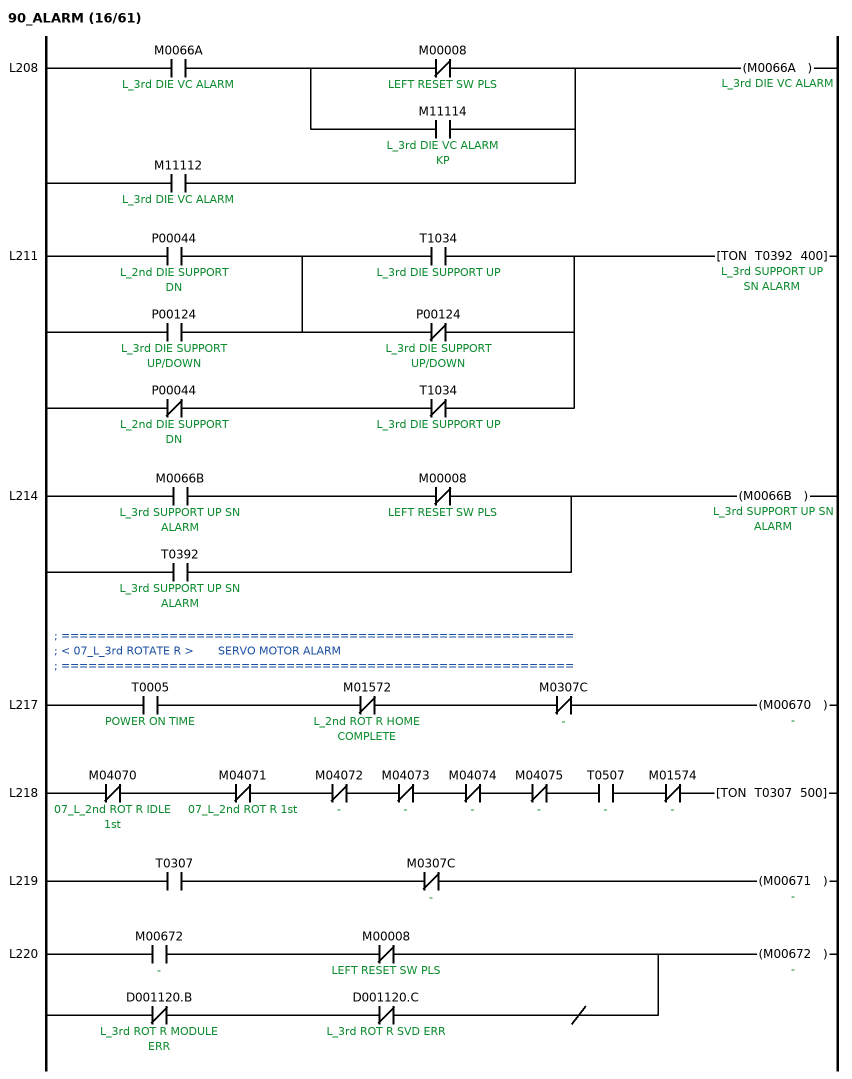
[picture p384: 90_ALARM rungs L208-L220]
; L208
LOAD      M0066A	// L_3rd DIE VC ALARM
LOAD NOT  M00008	// LEFT RESET SW PLS
OR        M11114	// L_3rd DIE VC ALARM KP
AND LOAD
OR        M11112	// L_3rd DIE VC ALARM
OUT       M0066A	// L_3rd DIE VC ALARM
; L211
LOAD      P00044	// L_2nd DIE SUPPORT DN
OR        P00124	// L_3rd DIE SUPPORT UP/DOWN
LOAD      T1034	// L_3rd DIE SUPPORT UP
OR NOT    P00124	// L_3rd DIE SUPPORT UP/DOWN
AND LOAD
LOAD NOT  P00044	// L_2nd DIE SUPPORT DN
AND NOT   T1034	// L_3rd DIE SUPPORT UP
OR LOAD
TON       T0392 400	// L_3rd SUPPORT UP SN ALARM
; L214
LOAD      M0066B	// L_3rd SUPPORT UP SN ALARM
AND NOT   M00008	// LEFT RESET SW PLS
OR        T0392	// L_3rd SUPPORT UP SN ALARM
OUT       M0066B	// L_3rd SUPPORT UP SN ALARM
// =========================================================
// 
//        < 07_L_3rd ROTATE R >       SERVO MOTOR ALARM
// 
// =========================================================
; L217
LOAD      T0005	// POWER ON TIME
AND NOT   M01572	// L_2nd ROT R HOME COMPLETE
AND NOT   M0307C	// -
OUT       M00670	// -
; L218
LOAD NOT  M04070	// 07_L_2nd ROT R IDLE 1st
AND NOT   M04071	// 07_L_2nd ROT R 1st
AND NOT   M04072	// -
AND NOT   M04073	// -
AND NOT   M04074	// -
AND NOT   M04075	// -
AND       T0507	// -
AND NOT   M01574	// -
TON       T0307 500
; L219
LOAD      T0307
AND NOT   M0307C	// -
OUT       M00671	// -
; L220
LOAD      M00672	// -
AND NOT   M00008	// LEFT RESET SW PLS
LOAD NOT  D001120.B	// L_3rd ROT R MODULE ERR
AND NOT   D001120.C	// L_3rd ROT R SVD ERR
NOT
OR LOAD
OUT       M00672	// -

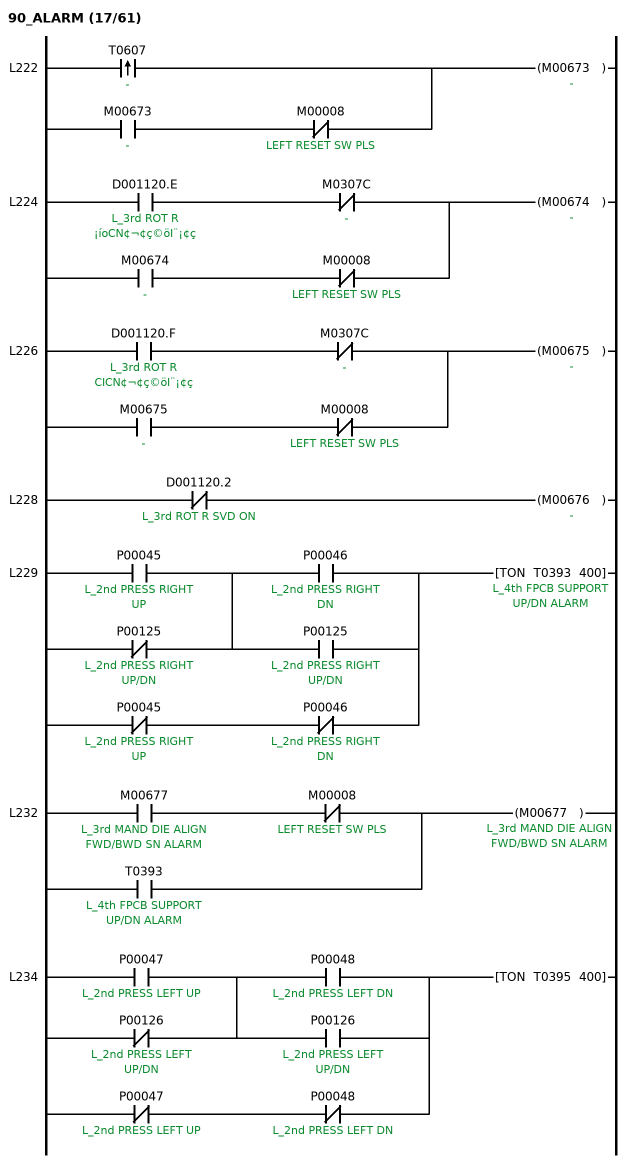
; L222
LOADP     T0607	// -
LOAD      M00673	// -
AND NOT   M00008	// LEFT RESET SW PLS
OR LOAD
OUT       M00673	// -
; L224
LOAD      D001120.E	// L_3rd ROT R ¡íoCN¢¬¢ç©öI¨¡¢ç
AND NOT   M0307C	// -
LOAD      M00674	// -
AND NOT   M00008	// LEFT RESET SW PLS
OR LOAD
OUT       M00674	// -
; L226
LOAD      D001120.F	// L_3rd ROT R CICN¢¬¢ç©öI¨¡¢ç
AND NOT   M0307C	// -
LOAD      M00675	// -
AND NOT   M00008	// LEFT RESET SW PLS
OR LOAD
OUT       M00675	// -
; L228
LOAD NOT  D001120.2	// L_3rd ROT R SVD ON
OUT       M00676	// -
; L229
LOAD      P00045	// L_2nd PRESS RIGHT UP
OR NOT    P00125	// L_2nd PRESS RIGHT UP/DN
LOAD      P00046	// L_2nd PRESS RIGHT DN
OR        P00125	// L_2nd PRESS RIGHT UP/DN
AND LOAD
LOAD NOT  P00045	// L_2nd PRESS RIGHT UP
AND NOT   P00046	// L_2nd PRESS RIGHT DN
OR LOAD
TON       T0393 400	// L_4th FPCB SUPPORT UP/DN ALARM
; L232
LOAD      M00677	// L_3rd MAND DIE ALIGN FWD/BWD SN ALARM
AND NOT   M00008	// LEFT RESET SW PLS
OR        T0393	// L_4th FPCB SUPPORT UP/DN ALARM
OUT       M00677	// L_3rd MAND DIE ALIGN FWD/BWD SN ALARM
; L234
LOAD      P00047	// L_2nd PRESS LEFT UP
OR NOT    P00126	// L_2nd PRESS LEFT UP/DN
LOAD      P00048	// L_2nd PRESS LEFT DN
OR        P00126	// L_2nd PRESS LEFT UP/DN
AND LOAD
LOAD NOT  P00047	// L_2nd PRESS LEFT UP
AND NOT   P00048	// L_2nd PRESS LEFT DN
OR LOAD
TON       T0395 400

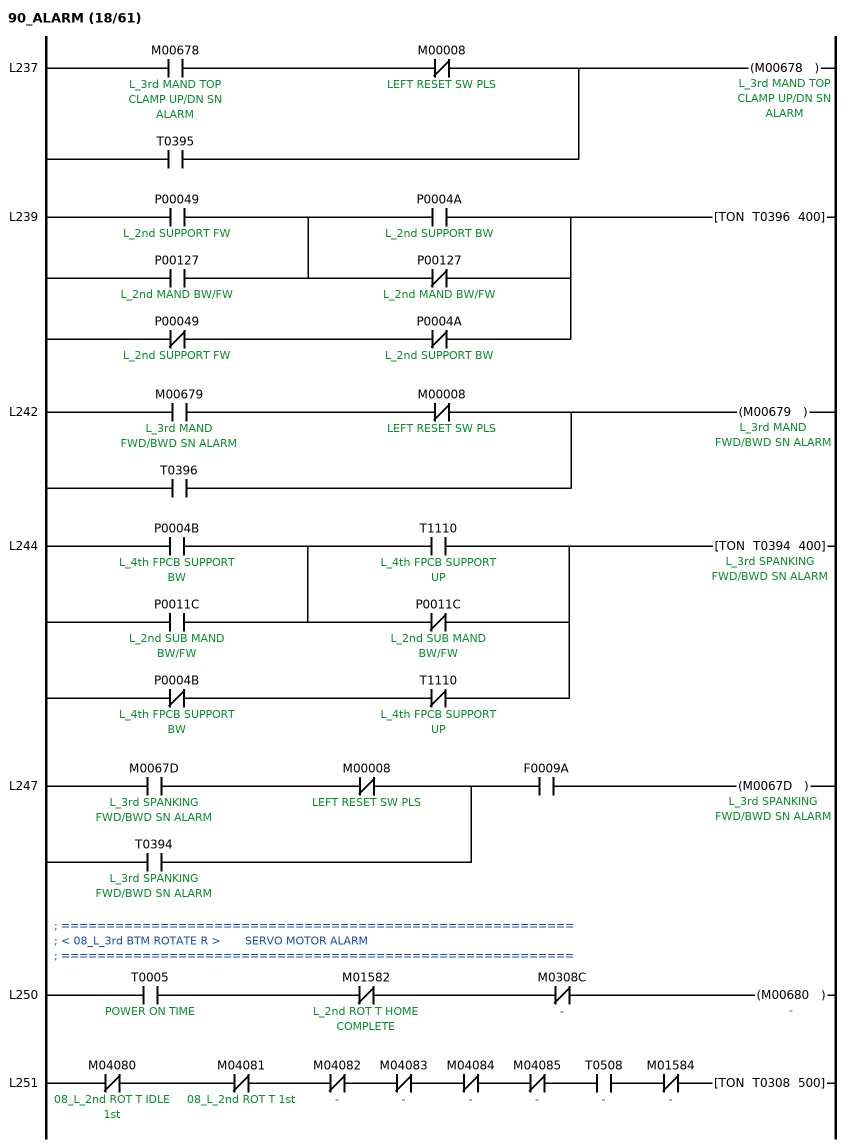
; L237
LOAD      M00678	// L_3rd MAND TOP CLAMP UP/DN SN ALARM
AND NOT   M00008	// LEFT RESET SW PLS
OR        T0395
OUT       M00678	// L_3rd MAND TOP CLAMP UP/DN SN ALARM
; L239
LOAD      P00049	// L_2nd SUPPORT FW
OR        P00127	// L_2nd MAND BW/FW
LOAD      P0004A	// L_2nd SUPPORT BW
OR NOT    P00127	// L_2nd MAND BW/FW
AND LOAD
LOAD NOT  P00049	// L_2nd SUPPORT FW
AND NOT   P0004A	// L_2nd SUPPORT BW
OR LOAD
TON       T0396 400
; L242
LOAD      M00679	// L_3rd MAND FWD/BWD SN ALARM
AND NOT   M00008	// LEFT RESET SW PLS
OR        T0396
OUT       M00679	// L_3rd MAND FWD/BWD SN ALARM
; L244
LOAD      P0004B	// L_4th FPCB SUPPORT BW
OR        P0011C	// L_2nd SUB MAND BW/FW
LOAD      T1110	// L_4th FPCB SUPPORT UP
OR NOT    P0011C	// L_2nd SUB MAND BW/FW
AND LOAD
LOAD NOT  P0004B	// L_4th FPCB SUPPORT BW
AND NOT   T1110	// L_4th FPCB SUPPORT UP
OR LOAD
TON       T0394 400	// L_3rd SPANKING FWD/BWD SN ALARM
; L247
LOAD      M0067D	// L_3rd SPANKING FWD/BWD SN ALARM
AND NOT   M00008	// LEFT RESET SW PLS
OR        T0394	// L_3rd SPANKING FWD/BWD SN ALARM
AND       F0009A
OUT       M0067D	// L_3rd SPANKING FWD/BWD SN ALARM
// =========================================================
// 
//        < 08_L_3rd BTM ROTATE R >       SERVO MOTOR ALARM
// 
// =========================================================
; L250
LOAD      T0005	// POWER ON TIME
AND NOT   M01582	// L_2nd ROT T HOME COMPLETE
AND NOT   M0308C	// -
OUT       M00680	// -
; L251
LOAD NOT  M04080	// 08_L_2nd ROT T IDLE 1st
AND NOT   M04081	// 08_L_2nd ROT T 1st
AND NOT   M04082	// -
AND NOT   M04083	// -
AND NOT   M04084	// -
AND NOT   M04085	// -
AND       T0508	// -
AND NOT   M01584	// -
TON       T0308 500

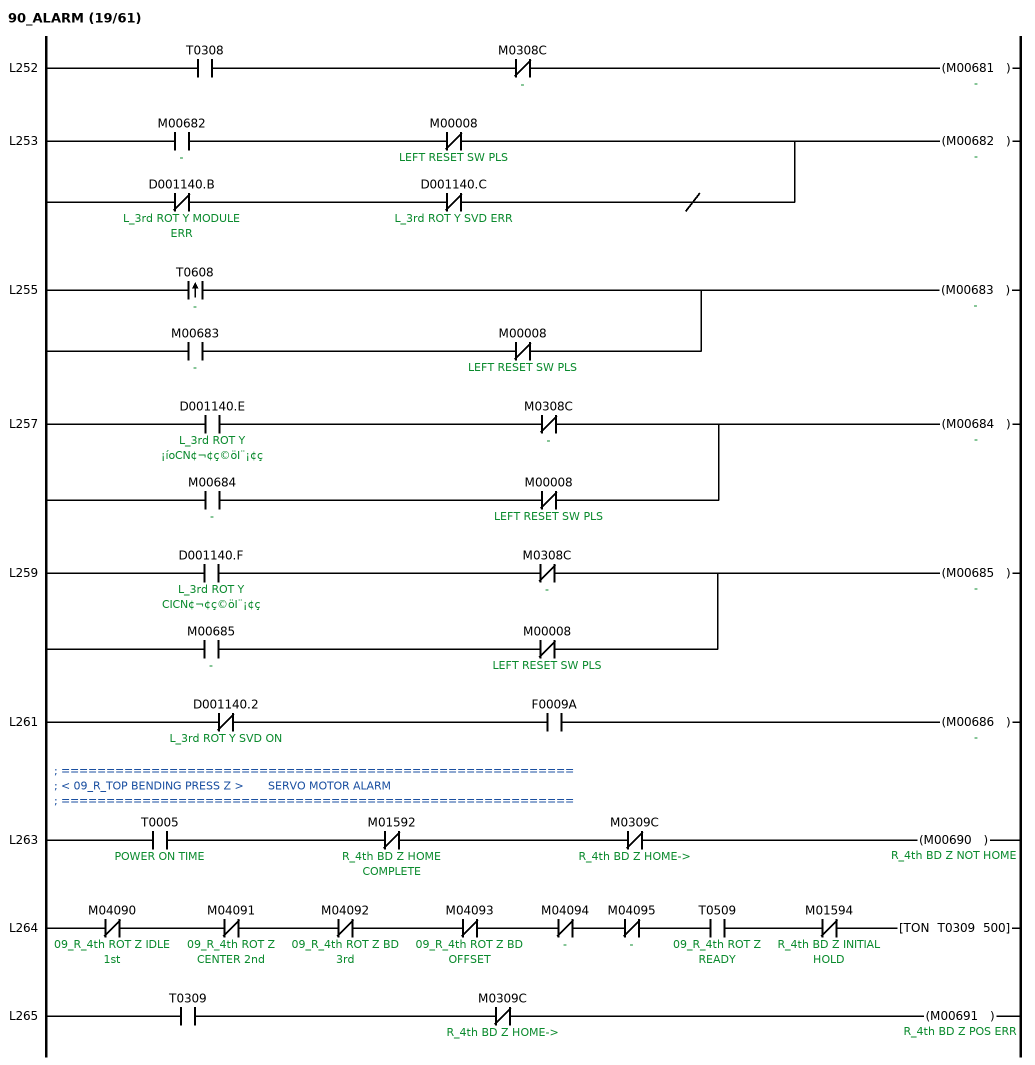
; L252
LOAD      T0308
AND NOT   M0308C	// -
OUT       M00681	// -
; L253
LOAD      M00682	// -
AND NOT   M00008	// LEFT RESET SW PLS
LOAD NOT  D001140.B	// L_3rd ROT Y MODULE ERR
AND NOT   D001140.C	// L_3rd ROT Y SVD ERR
NOT
OR LOAD
OUT       M00682	// -
; L255
LOADP     T0608	// -
LOAD      M00683	// -
AND NOT   M00008	// LEFT RESET SW PLS
OR LOAD
OUT       M00683	// -
; L257
LOAD      D001140.E	// L_3rd ROT Y ¡íoCN¢¬¢ç©öI¨¡¢ç
AND NOT   M0308C	// -
LOAD      M00684	// -
AND NOT   M00008	// LEFT RESET SW PLS
OR LOAD
OUT       M00684	// -
; L259
LOAD      D001140.F	// L_3rd ROT Y CICN¢¬¢ç©öI¨¡¢ç
AND NOT   M0308C	// -
LOAD      M00685	// -
AND NOT   M00008	// LEFT RESET SW PLS
OR LOAD
OUT       M00685	// -
; L261
LOAD NOT  D001140.2	// L_3rd ROT Y SVD ON
AND       F0009A
OUT       M00686	// -
// =========================================================
// 
//        < 09_R_TOP BENDING PRESS Z >       SERVO MOTOR ALARM
// 
// =========================================================
; L263
LOAD      T0005	// POWER ON TIME
AND NOT   M01592	// R_4th BD Z HOME COMPLETE
AND NOT   M0309C	// R_4th BD Z HOME->
OUT       M00690	// R_4th BD Z NOT HOME
; L264
LOAD NOT  M04090	// 09_R_4th ROT Z IDLE 1st
AND NOT   M04091	// 09_R_4th ROT Z CENTER 2nd
AND NOT   M04092	// 09_R_4th ROT Z BD 3rd
AND NOT   M04093	// 09_R_4th ROT Z BD OFFSET
AND NOT   M04094	// -
AND NOT   M04095	// -
AND       T0509	// 09_R_4th ROT Z READY
AND NOT   M01594	// R_4th BD Z INITIAL HOLD
TON       T0309 500
; L265
LOAD      T0309
AND NOT   M0309C	// R_4th BD Z HOME->
OUT       M00691	// R_4th BD Z POS ERR

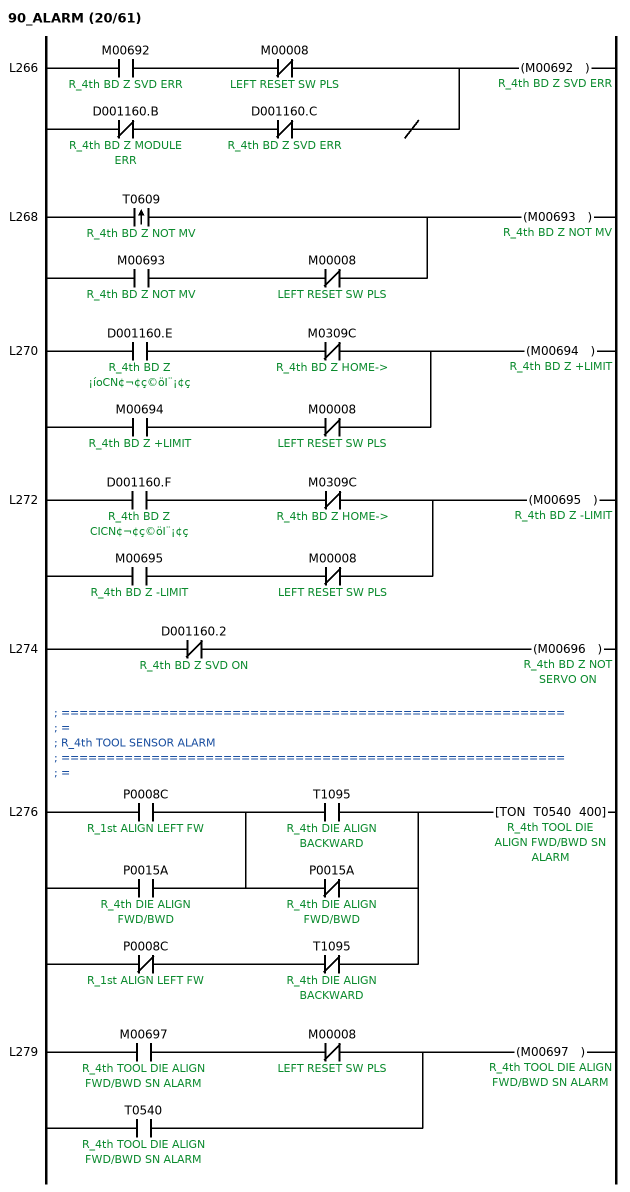
; L266
LOAD      M00692	// R_4th BD Z SVD ERR
AND NOT   M00008	// LEFT RESET SW PLS
LOAD NOT  D001160.B	// R_4th BD Z MODULE ERR
AND NOT   D001160.C	// R_4th BD Z SVD ERR
NOT
OR LOAD
OUT       M00692	// R_4th BD Z SVD ERR
; L268
LOADP     T0609	// R_4th BD Z NOT MV
LOAD      M00693	// R_4th BD Z NOT MV
AND NOT   M00008	// LEFT RESET SW PLS
OR LOAD
OUT       M00693	// R_4th BD Z NOT MV
; L270
LOAD      D001160.E	// R_4th BD Z ¡íoCN¢¬¢ç©öI¨¡¢ç
AND NOT   M0309C	// R_4th BD Z HOME->
LOAD      M00694	// R_4th BD Z +LIMIT
AND NOT   M00008	// LEFT RESET SW PLS
OR LOAD
OUT       M00694	// R_4th BD Z +LIMIT
; L272
LOAD      D001160.F	// R_4th BD Z CICN¢¬¢ç©öI¨¡¢ç
AND NOT   M0309C	// R_4th BD Z HOME->
LOAD      M00695	// R_4th BD Z -LIMIT
AND NOT   M00008	// LEFT RESET SW PLS
OR LOAD
OUT       M00695	// R_4th BD Z -LIMIT
; L274
LOAD NOT  D001160.2	// R_4th BD Z SVD ON
OUT       M00696	// R_4th BD Z NOT SERVO ON
// =========================================================
// 
//        R_4th TOOL SENSOR ALARM
// 
// =========================================================
; L276
LOAD      P0008C	// R_1st ALIGN LEFT FW
OR        P0015A	// R_4th DIE ALIGN FWD/BWD
LOAD      T1095	// R_4th DIE ALIGN BACKWARD
OR NOT    P0015A	// R_4th DIE ALIGN FWD/BWD
AND LOAD
LOAD NOT  P0008C	// R_1st ALIGN LEFT FW
AND NOT   T1095	// R_4th DIE ALIGN BACKWARD
OR LOAD
TON       T0540 400	// R_4th TOOL DIE ALIGN FWD/BWD SN ALARM
; L279
LOAD      M00697	// R_4th TOOL DIE ALIGN FWD/BWD SN ALARM
AND NOT   M00008	// LEFT RESET SW PLS
OR        T0540	// R_4th TOOL DIE ALIGN FWD/BWD SN ALARM
OUT       M00697	// R_4th TOOL DIE ALIGN FWD/BWD SN ALARM

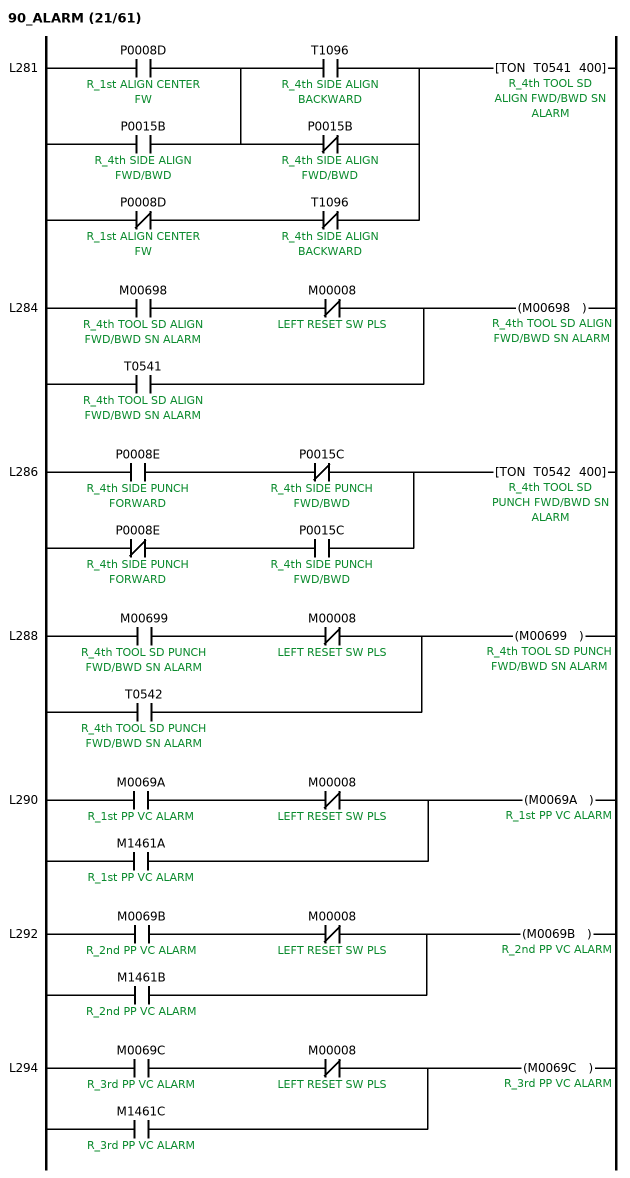
; L281
LOAD      P0008D	// R_1st ALIGN CENTER FW
OR        P0015B	// R_4th SIDE ALIGN FWD/BWD
LOAD      T1096	// R_4th SIDE ALIGN BACKWARD
OR NOT    P0015B	// R_4th SIDE ALIGN FWD/BWD
AND LOAD
LOAD NOT  P0008D	// R_1st ALIGN CENTER FW
AND NOT   T1096	// R_4th SIDE ALIGN BACKWARD
OR LOAD
TON       T0541 400	// R_4th TOOL SD ALIGN FWD/BWD SN ALARM
; L284
LOAD      M00698	// R_4th TOOL SD ALIGN FWD/BWD SN ALARM
AND NOT   M00008	// LEFT RESET SW PLS
OR        T0541	// R_4th TOOL SD ALIGN FWD/BWD SN ALARM
OUT       M00698	// R_4th TOOL SD ALIGN FWD/BWD SN ALARM
; L286
LOAD      P0008E	// R_4th SIDE PUNCH FORWARD
AND NOT   P0015C	// R_4th SIDE PUNCH FWD/BWD
LOAD NOT  P0008E	// R_4th SIDE PUNCH FORWARD
AND       P0015C	// R_4th SIDE PUNCH FWD/BWD
OR LOAD
TON       T0542 400	// R_4th TOOL SD PUNCH FWD/BWD SN ALARM
; L288
LOAD      M00699	// R_4th TOOL SD PUNCH FWD/BWD SN ALARM
AND NOT   M00008	// LEFT RESET SW PLS
OR        T0542	// R_4th TOOL SD PUNCH FWD/BWD SN ALARM
OUT       M00699	// R_4th TOOL SD PUNCH FWD/BWD SN ALARM
; L290
LOAD      M0069A	// R_1st PP VC ALARM
AND NOT   M00008	// LEFT RESET SW PLS
OR        M1461A	// R_1st PP VC ALARM
OUT       M0069A	// R_1st PP VC ALARM
; L292
LOAD      M0069B	// R_2nd PP VC ALARM
AND NOT   M00008	// LEFT RESET SW PLS
OR        M1461B	// R_2nd PP VC ALARM
OUT       M0069B	// R_2nd PP VC ALARM
; L294
LOAD      M0069C	// R_3rd PP VC ALARM
AND NOT   M00008	// LEFT RESET SW PLS
OR        M1461C	// R_3rd PP VC ALARM
OUT       M0069C	// R_3rd PP VC ALARM

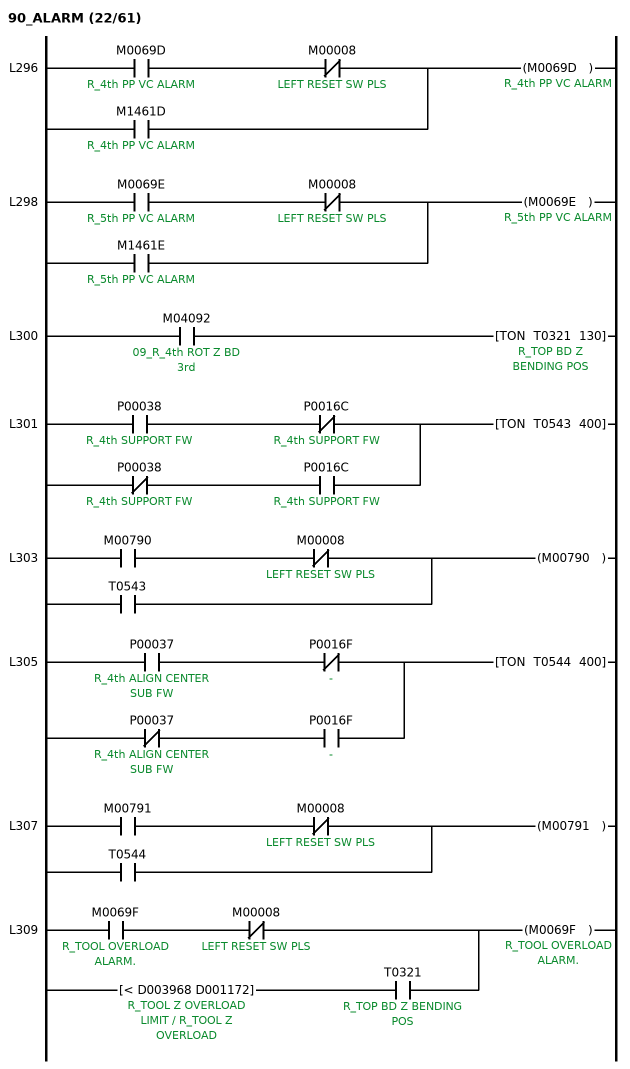
; L296
LOAD      M0069D	// R_4th PP VC ALARM
AND NOT   M00008	// LEFT RESET SW PLS
OR        M1461D	// R_4th PP VC ALARM
OUT       M0069D	// R_4th PP VC ALARM
; L298
LOAD      M0069E	// R_5th PP VC ALARM
AND NOT   M00008	// LEFT RESET SW PLS
OR        M1461E	// R_5th PP VC ALARM
OUT       M0069E	// R_5th PP VC ALARM
; L300
LOAD      M04092	// 09_R_4th ROT Z BD 3rd
TON       T0321 130	// R_TOP BD Z BENDING POS
; L301
LOAD      P00038	// R_4th SUPPORT FW
AND NOT   P0016C	// R_4th SUPPORT FW
LOAD NOT  P00038	// R_4th SUPPORT FW
AND       P0016C	// R_4th SUPPORT FW
OR LOAD
TON       T0543 400
; L303
LOAD      M00790
AND NOT   M00008	// LEFT RESET SW PLS
OR        T0543
OUT       M00790
; L305
LOAD      P00037	// R_4th ALIGN CENTER SUB FW
AND NOT   P0016F	// -
LOAD NOT  P00037	// R_4th ALIGN CENTER SUB FW
AND       P0016F	// -
OR LOAD
TON       T0544 400
; L307
LOAD      M00791
AND NOT   M00008	// LEFT RESET SW PLS
OR        T0544
OUT       M00791
; L309
LOAD      M0069F	// R_TOOL OVERLOAD ALARM.
AND NOT   M00008	// LEFT RESET SW PLS
LOAD<     D003968 D001172	// R_TOOL Z OVERLOAD LIMIT / R_TOOL Z OVERLOAD
AND       T0321	// R_TOP BD Z BENDING POS
OR LOAD
OUT       M0069F	// R_TOOL OVERLOAD ALARM.

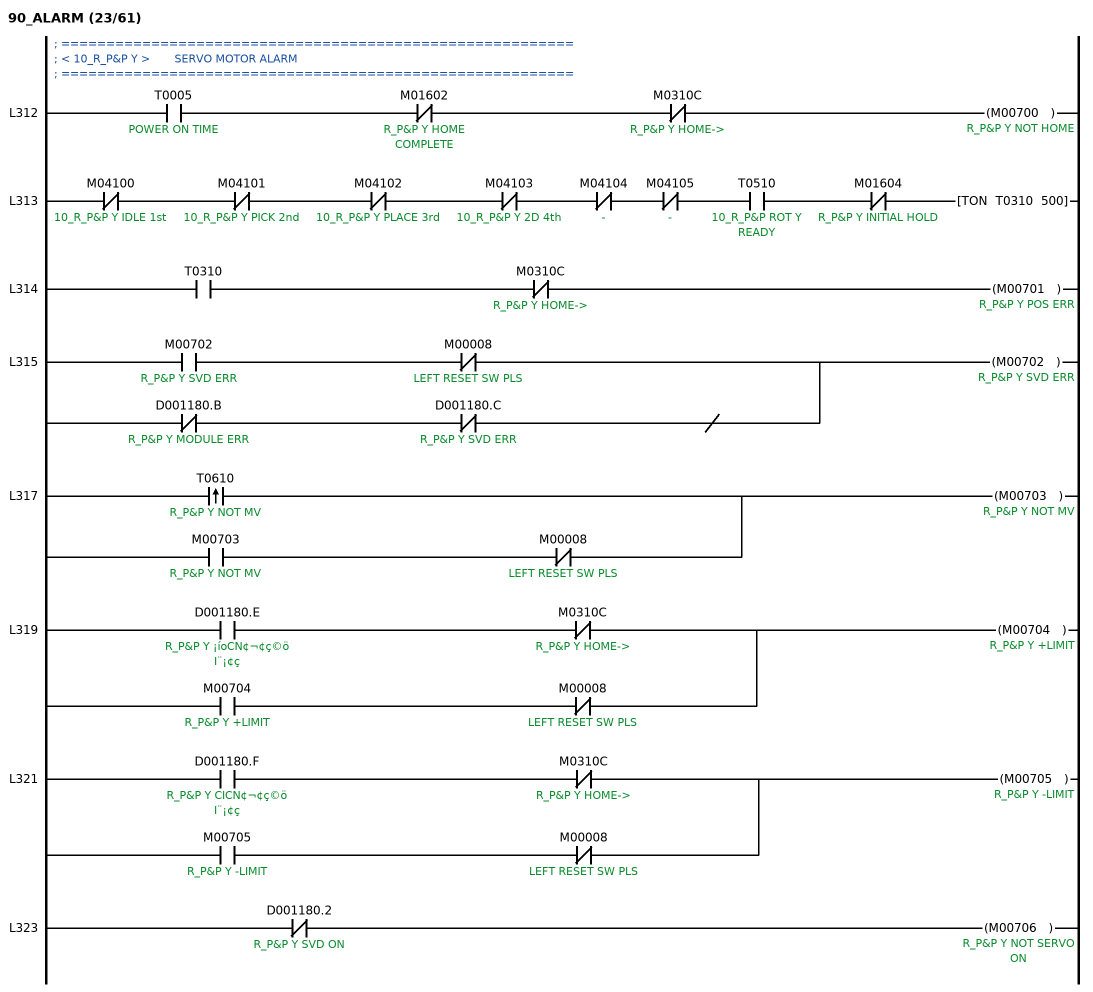
// =========================================================
// 
//        < 10_R_P&P Y >       SERVO MOTOR ALARM
// 
// =========================================================
; L312
LOAD      T0005	// POWER ON TIME
AND NOT   M01602	// R_P&P Y HOME COMPLETE
AND NOT   M0310C	// R_P&P Y HOME->
OUT       M00700	// R_P&P Y NOT HOME
; L313
LOAD NOT  M04100	// 10_R_P&P Y IDLE 1st
AND NOT   M04101	// 10_R_P&P Y PICK 2nd
AND NOT   M04102	// 10_R_P&P Y PLACE 3rd
AND NOT   M04103	// 10_R_P&P Y 2D 4th
AND NOT   M04104	// -
AND NOT   M04105	// -
AND       T0510	// 10_R_P&P ROT Y READY
AND NOT   M01604	// R_P&P Y INITIAL HOLD
TON       T0310 500
; L314
LOAD      T0310
AND NOT   M0310C	// R_P&P Y HOME->
OUT       M00701	// R_P&P Y POS ERR
; L315
LOAD      M00702	// R_P&P Y SVD ERR
AND NOT   M00008	// LEFT RESET SW PLS
LOAD NOT  D001180.B	// R_P&P Y MODULE ERR
AND NOT   D001180.C	// R_P&P Y SVD ERR
NOT
OR LOAD
OUT       M00702	// R_P&P Y SVD ERR
; L317
LOADP     T0610	// R_P&P Y NOT MV
LOAD      M00703	// R_P&P Y NOT MV
AND NOT   M00008	// LEFT RESET SW PLS
OR LOAD
OUT       M00703	// R_P&P Y NOT MV
; L319
LOAD      D001180.E	// R_P&P Y ¡íoCN¢¬¢ç©öI¨¡¢ç
AND NOT   M0310C	// R_P&P Y HOME->
LOAD      M00704	// R_P&P Y +LIMIT
AND NOT   M00008	// LEFT RESET SW PLS
OR LOAD
OUT       M00704	// R_P&P Y +LIMIT
; L321
LOAD      D001180.F	// R_P&P Y CICN¢¬¢ç©öI¨¡¢ç
AND NOT   M0310C	// R_P&P Y HOME->
LOAD      M00705	// R_P&P Y -LIMIT
AND NOT   M00008	// LEFT RESET SW PLS
OR LOAD
OUT       M00705	// R_P&P Y -LIMIT
; L323
LOAD NOT  D001180.2	// R_P&P Y SVD ON
OUT       M00706	// R_P&P Y NOT SERVO ON

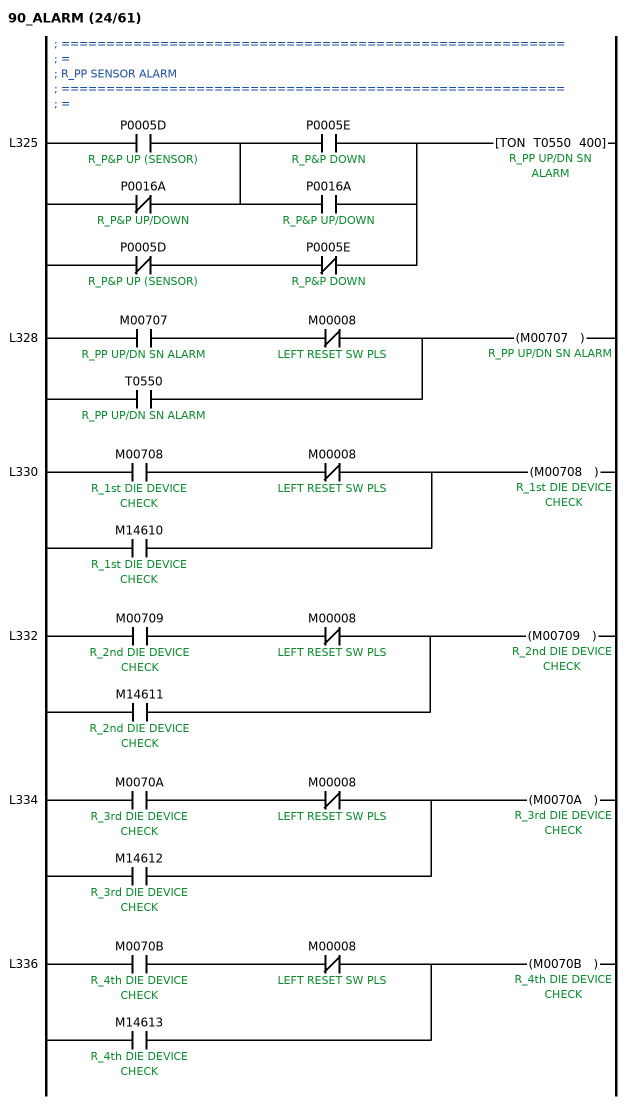
// =========================================================
// 
//       R_PP SENSOR ALARM
// 
// =========================================================
; L325
LOAD      P0005D	// R_P&P UP (SENSOR)
OR NOT    P0016A	// R_P&P UP/DOWN
LOAD      P0005E	// R_P&P DOWN
OR        P0016A	// R_P&P UP/DOWN
AND LOAD
LOAD NOT  P0005D	// R_P&P UP (SENSOR)
AND NOT   P0005E	// R_P&P DOWN
OR LOAD
TON       T0550 400	// R_PP UP/DN SN ALARM
; L328
LOAD      M00707	// R_PP UP/DN SN ALARM
AND NOT   M00008	// LEFT RESET SW PLS
OR        T0550	// R_PP UP/DN SN ALARM
OUT       M00707	// R_PP UP/DN SN ALARM
; L330
LOAD      M00708	// R_1st DIE DEVICE CHECK
AND NOT   M00008	// LEFT RESET SW PLS
OR        M14610	// R_1st DIE DEVICE CHECK
OUT       M00708	// R_1st DIE DEVICE CHECK
; L332
LOAD      M00709	// R_2nd DIE DEVICE CHECK
AND NOT   M00008	// LEFT RESET SW PLS
OR        M14611	// R_2nd DIE DEVICE CHECK
OUT       M00709	// R_2nd DIE DEVICE CHECK
; L334
LOAD      M0070A	// R_3rd DIE DEVICE CHECK
AND NOT   M00008	// LEFT RESET SW PLS
OR        M14612	// R_3rd DIE DEVICE CHECK
OUT       M0070A	// R_3rd DIE DEVICE CHECK
; L336
LOAD      M0070B	// R_4th DIE DEVICE CHECK
AND NOT   M00008	// LEFT RESET SW PLS
OR        M14613	// R_4th DIE DEVICE CHECK
OUT       M0070B	// R_4th DIE DEVICE CHECK

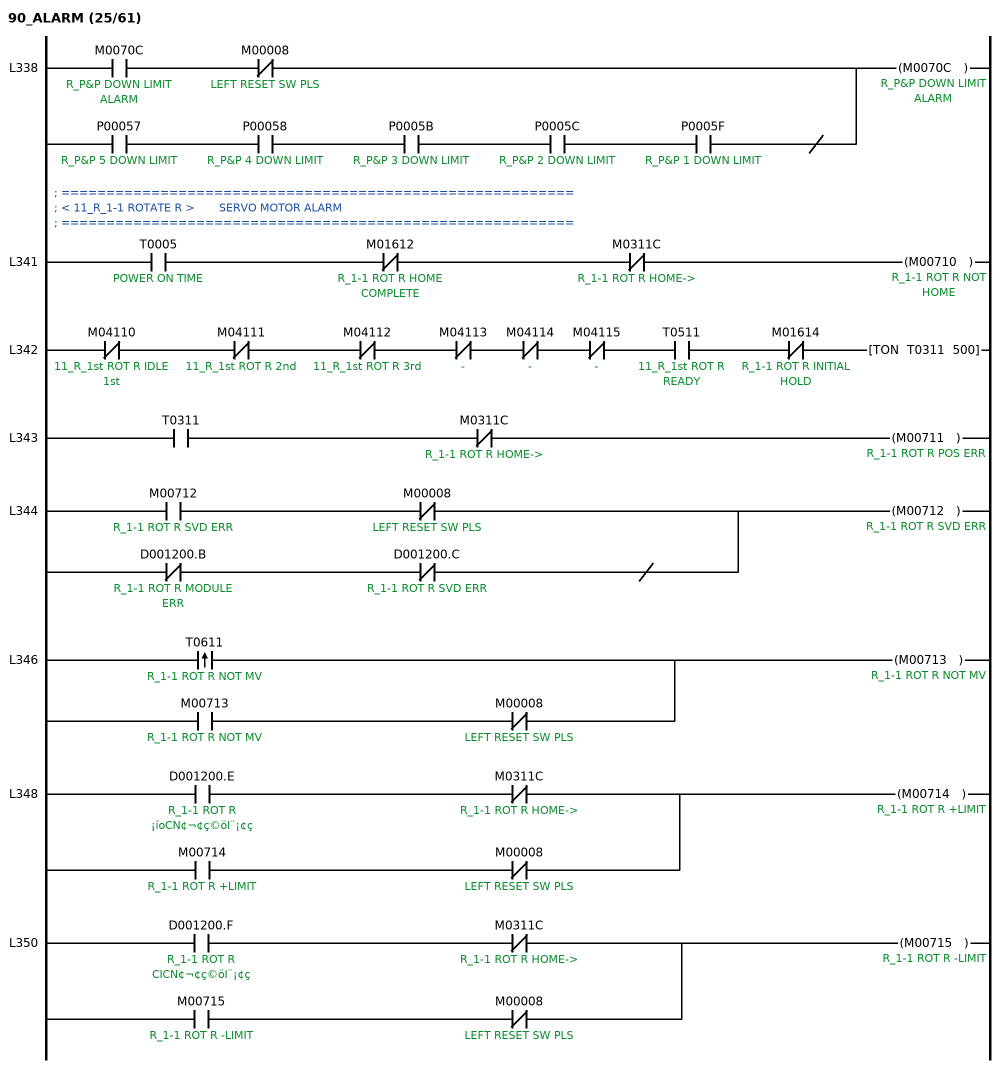
; L338
LOAD      M0070C	// R_P&P DOWN LIMIT ALARM
AND NOT   M00008	// LEFT RESET SW PLS
LOAD      P00057	// R_P&P 5 DOWN LIMIT
AND       P00058	// R_P&P 4 DOWN LIMIT
AND       P0005B	// R_P&P 3 DOWN LIMIT
AND       P0005C	// R_P&P 2 DOWN LIMIT
AND       P0005F	// R_P&P 1 DOWN LIMIT
NOT
OR LOAD
OUT       M0070C	// R_P&P DOWN LIMIT ALARM
// =========================================================
// 
//        < 11_R_1-1 ROTATE R >       SERVO MOTOR ALARM
// 
// =========================================================
; L341
LOAD      T0005	// POWER ON TIME
AND NOT   M01612	// R_1-1 ROT R HOME COMPLETE
AND NOT   M0311C	// R_1-1 ROT R HOME->
OUT       M00710	// R_1-1 ROT R NOT HOME
; L342
LOAD NOT  M04110	// 11_R_1st ROT R IDLE 1st
AND NOT   M04111	// 11_R_1st ROT R 2nd
AND NOT   M04112	// 11_R_1st ROT R 3rd
AND NOT   M04113	// -
AND NOT   M04114	// -
AND NOT   M04115	// -
AND       T0511	// 11_R_1st ROT R READY
AND NOT   M01614	// R_1-1 ROT R INITIAL HOLD
TON       T0311 500
; L343
LOAD      T0311
AND NOT   M0311C	// R_1-1 ROT R HOME->
OUT       M00711	// R_1-1 ROT R POS ERR
; L344
LOAD      M00712	// R_1-1 ROT R SVD ERR
AND NOT   M00008	// LEFT RESET SW PLS
LOAD NOT  D001200.B	// R_1-1 ROT R MODULE ERR
AND NOT   D001200.C	// R_1-1 ROT R SVD ERR
NOT
OR LOAD
OUT       M00712	// R_1-1 ROT R SVD ERR
; L346
LOADP     T0611	// R_1-1 ROT R NOT MV
LOAD      M00713	// R_1-1 ROT R NOT MV
AND NOT   M00008	// LEFT RESET SW PLS
OR LOAD
OUT       M00713	// R_1-1 ROT R NOT MV
; L348
LOAD      D001200.E	// R_1-1 ROT R ¡íoCN¢¬¢ç©öI¨¡¢ç
AND NOT   M0311C	// R_1-1 ROT R HOME->
LOAD      M00714	// R_1-1 ROT R +LIMIT
AND NOT   M00008	// LEFT RESET SW PLS
OR LOAD
OUT       M00714	// R_1-1 ROT R +LIMIT
; L350
LOAD      D001200.F	// R_1-1 ROT R CICN¢¬¢ç©öI¨¡¢ç
AND NOT   M0311C	// R_1-1 ROT R HOME->
LOAD      M00715	// R_1-1 ROT R -LIMIT
AND NOT   M00008	// LEFT RESET SW PLS
OR LOAD
OUT       M00715	// R_1-1 ROT R -LIMIT

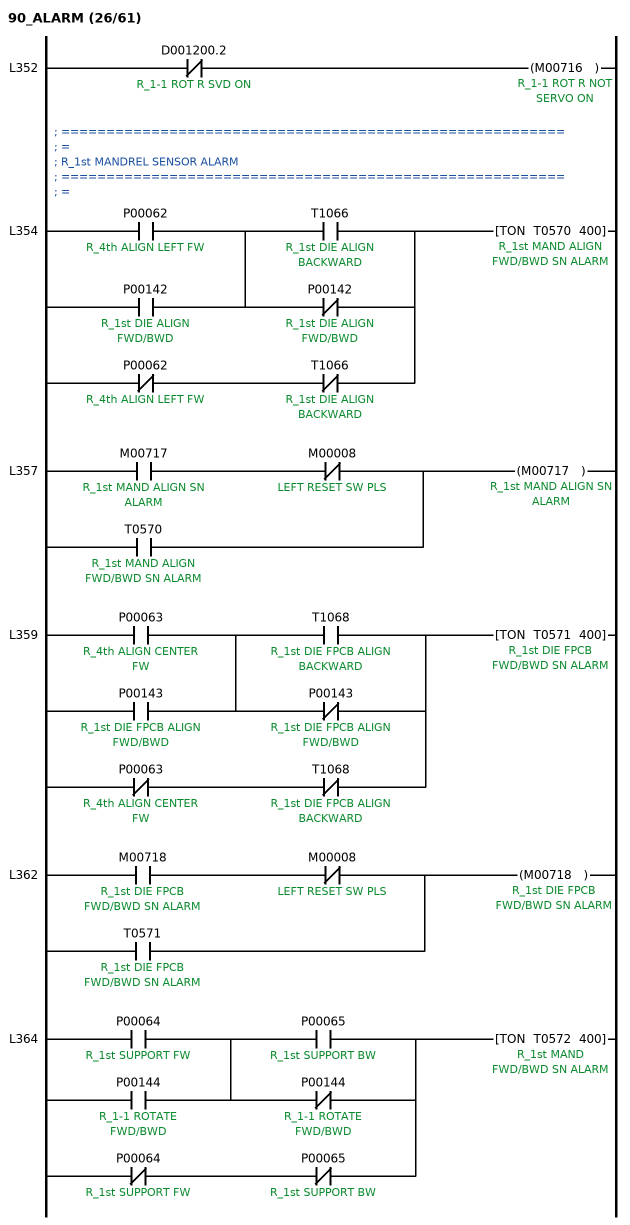
; L352
LOAD NOT  D001200.2	// R_1-1 ROT R SVD ON
OUT       M00716	// R_1-1 ROT R NOT SERVO ON
// =========================================================
// 
//        R_1st MANDREL SENSOR ALARM
// 
// =========================================================
; L354
LOAD      P00062	// R_4th ALIGN LEFT FW
OR        P00142	// R_1st DIE ALIGN FWD/BWD
LOAD      T1066	// R_1st DIE ALIGN BACKWARD
OR NOT    P00142	// R_1st DIE ALIGN FWD/BWD
AND LOAD
LOAD NOT  P00062	// R_4th ALIGN LEFT FW
AND NOT   T1066	// R_1st DIE ALIGN BACKWARD
OR LOAD
TON       T0570 400	// R_1st MAND ALIGN FWD/BWD SN ALARM
; L357
LOAD      M00717	// R_1st MAND ALIGN SN ALARM
AND NOT   M00008	// LEFT RESET SW PLS
OR        T0570	// R_1st MAND ALIGN FWD/BWD SN ALARM
OUT       M00717	// R_1st MAND ALIGN SN ALARM
; L359
LOAD      P00063	// R_4th ALIGN CENTER FW
OR        P00143	// R_1st DIE FPCB ALIGN FWD/BWD
LOAD      T1068	// R_1st DIE FPCB ALIGN BACKWARD
OR NOT    P00143	// R_1st DIE FPCB ALIGN FWD/BWD
AND LOAD
LOAD NOT  P00063	// R_4th ALIGN CENTER FW
AND NOT   T1068	// R_1st DIE FPCB ALIGN BACKWARD
OR LOAD
TON       T0571 400	// R_1st DIE FPCB FWD/BWD SN ALARM
; L362
LOAD      M00718	// R_1st DIE FPCB FWD/BWD SN ALARM
AND NOT   M00008	// LEFT RESET SW PLS
OR        T0571	// R_1st DIE FPCB FWD/BWD SN ALARM
OUT       M00718	// R_1st DIE FPCB FWD/BWD SN ALARM
; L364
LOAD      P00064	// R_1st SUPPORT FW
OR        P00144	// R_1-1 ROTATE FWD/BWD
LOAD      P00065	// R_1st SUPPORT BW
OR NOT    P00144	// R_1-1 ROTATE FWD/BWD
AND LOAD
LOAD NOT  P00064	// R_1st SUPPORT FW
AND NOT   P00065	// R_1st SUPPORT BW
OR LOAD
TON       T0572 400	// R_1st MAND FWD/BWD SN ALARM

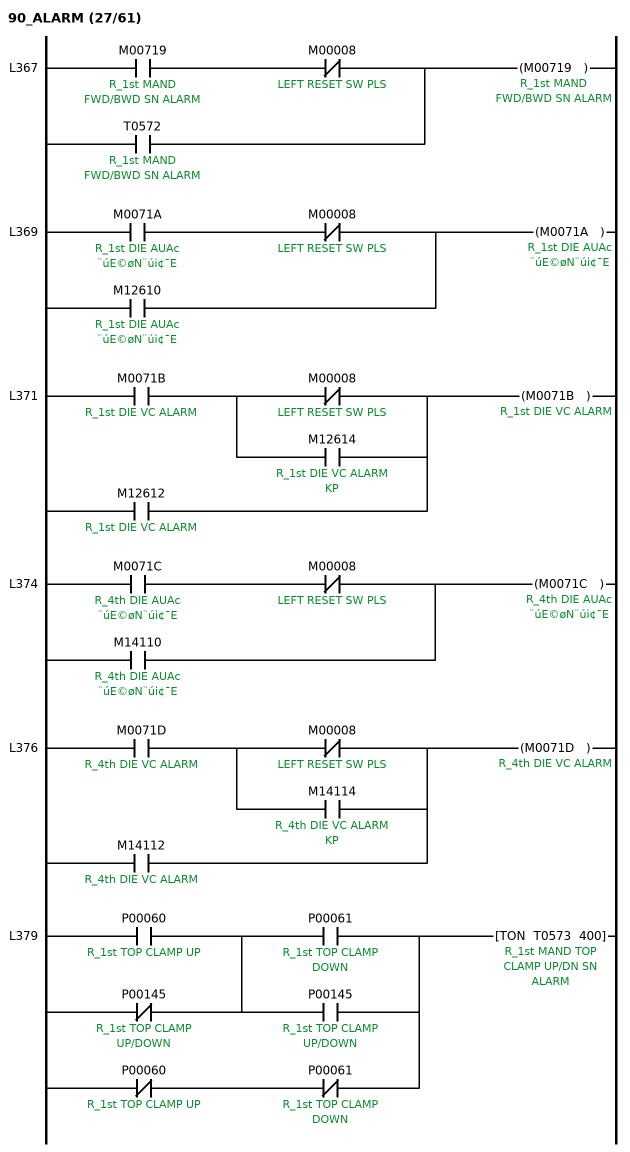
; L367
LOAD      M00719	// R_1st MAND FWD/BWD SN ALARM
AND NOT   M00008	// LEFT RESET SW PLS
OR        T0572	// R_1st MAND FWD/BWD SN ALARM
OUT       M00719	// R_1st MAND FWD/BWD SN ALARM
; L369
LOAD      M0071A	// R_1st DIE AUAc ¨úE©øN¨úi¢¯E
AND NOT   M00008	// LEFT RESET SW PLS
OR        M12610	// R_1st DIE AUAc ¨úE©øN¨úi¢¯E
OUT       M0071A	// R_1st DIE AUAc ¨úE©øN¨úi¢¯E
; L371
LOAD      M0071B	// R_1st DIE VC ALARM
LOAD NOT  M00008	// LEFT RESET SW PLS
OR        M12614	// R_1st DIE VC ALARM KP
AND LOAD
OR        M12612	// R_1st DIE VC ALARM
OUT       M0071B	// R_1st DIE VC ALARM
; L374
LOAD      M0071C	// R_4th DIE AUAc ¨úE©øN¨úi¢¯E
AND NOT   M00008	// LEFT RESET SW PLS
OR        M14110	// R_4th DIE AUAc ¨úE©øN¨úi¢¯E
OUT       M0071C	// R_4th DIE AUAc ¨úE©øN¨úi¢¯E
; L376
LOAD      M0071D	// R_4th DIE VC ALARM
LOAD NOT  M00008	// LEFT RESET SW PLS
OR        M14114	// R_4th DIE VC ALARM KP
AND LOAD
OR        M14112	// R_4th DIE VC ALARM
OUT       M0071D	// R_4th DIE VC ALARM
; L379
LOAD      P00060	// R_1st TOP CLAMP UP
OR NOT    P00145	// R_1st TOP CLAMP UP/DOWN
LOAD      P00061	// R_1st TOP CLAMP DOWN
OR        P00145	// R_1st TOP CLAMP UP/DOWN
AND LOAD
LOAD NOT  P00060	// R_1st TOP CLAMP UP
AND NOT   P00061	// R_1st TOP CLAMP DOWN
OR LOAD
TON       T0573 400	// R_1st MAND TOP CLAMP UP/DN SN ALARM

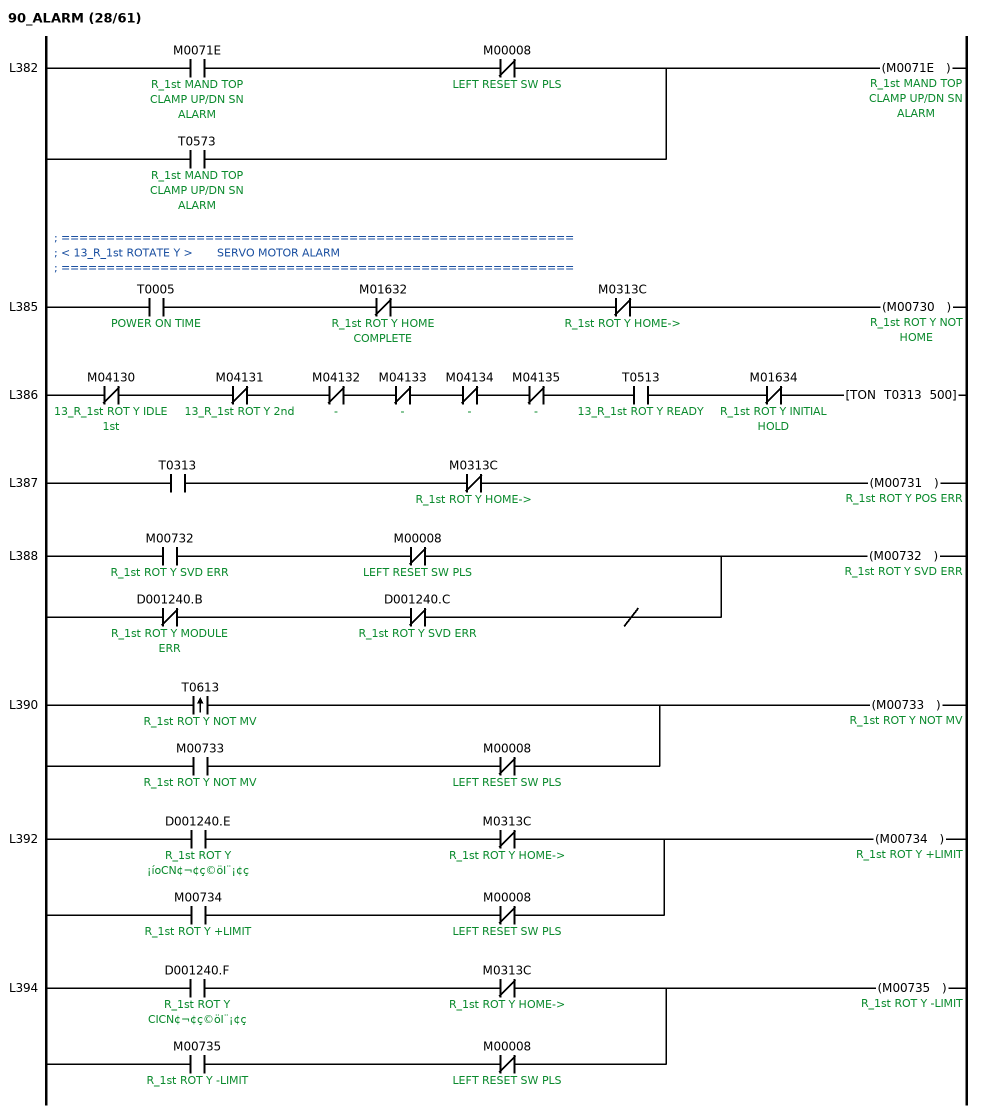
; L382
LOAD      M0071E	// R_1st MAND TOP CLAMP UP/DN SN ALARM
AND NOT   M00008	// LEFT RESET SW PLS
OR        T0573	// R_1st MAND TOP CLAMP UP/DN SN ALARM
OUT       M0071E	// R_1st MAND TOP CLAMP UP/DN SN ALARM
// =========================================================
// 
//        < 13_R_1st ROTATE Y >       SERVO MOTOR ALARM
// 
// =========================================================
; L385
LOAD      T0005	// POWER ON TIME
AND NOT   M01632	// R_1st ROT Y HOME COMPLETE
AND NOT   M0313C	// R_1st ROT Y HOME->
OUT       M00730	// R_1st ROT Y NOT HOME
; L386
LOAD NOT  M04130	// 13_R_1st ROT Y IDLE 1st
AND NOT   M04131	// 13_R_1st ROT Y 2nd
AND NOT   M04132	// -
AND NOT   M04133	// -
AND NOT   M04134	// -
AND NOT   M04135	// -
AND       T0513	// 13_R_1st ROT Y READY
AND NOT   M01634	// R_1st ROT Y INITIAL HOLD
TON       T0313 500
; L387
LOAD      T0313
AND NOT   M0313C	// R_1st ROT Y HOME->
OUT       M00731	// R_1st ROT Y POS ERR
; L388
LOAD      M00732	// R_1st ROT Y SVD ERR
AND NOT   M00008	// LEFT RESET SW PLS
LOAD NOT  D001240.B	// R_1st ROT Y MODULE ERR
AND NOT   D001240.C	// R_1st ROT Y SVD ERR
NOT
OR LOAD
OUT       M00732	// R_1st ROT Y SVD ERR
; L390
LOADP     T0613	// R_1st ROT Y NOT MV
LOAD      M00733	// R_1st ROT Y NOT MV
AND NOT   M00008	// LEFT RESET SW PLS
OR LOAD
OUT       M00733	// R_1st ROT Y NOT MV
; L392
LOAD      D001240.E	// R_1st ROT Y ¡íoCN¢¬¢ç©öI¨¡¢ç
AND NOT   M0313C	// R_1st ROT Y HOME->
LOAD      M00734	// R_1st ROT Y +LIMIT
AND NOT   M00008	// LEFT RESET SW PLS
OR LOAD
OUT       M00734	// R_1st ROT Y +LIMIT
; L394
LOAD      D001240.F	// R_1st ROT Y CICN¢¬¢ç©öI¨¡¢ç
AND NOT   M0313C	// R_1st ROT Y HOME->
LOAD      M00735	// R_1st ROT Y -LIMIT
AND NOT   M00008	// LEFT RESET SW PLS
OR LOAD
OUT       M00735	// R_1st ROT Y -LIMIT

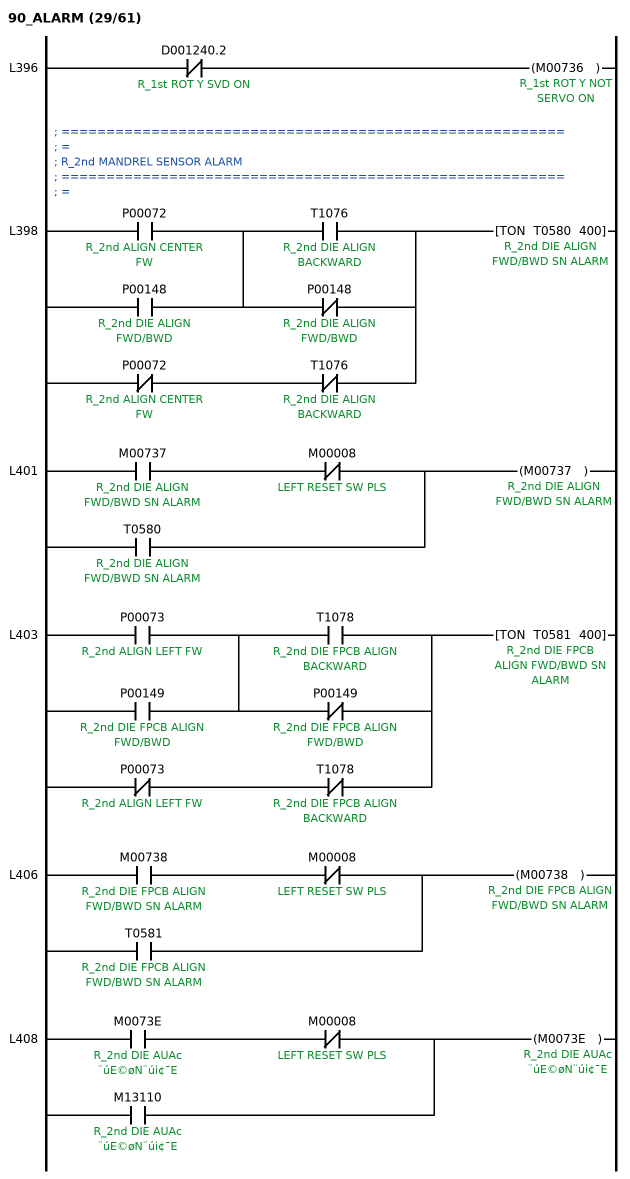
; L396
LOAD NOT  D001240.2	// R_1st ROT Y SVD ON
OUT       M00736	// R_1st ROT Y NOT SERVO ON
// =========================================================
// 
//        R_2nd MANDREL SENSOR ALARM
// 
// =========================================================
; L398
LOAD      P00072	// R_2nd ALIGN CENTER FW
OR        P00148	// R_2nd DIE ALIGN FWD/BWD
LOAD      T1076	// R_2nd DIE ALIGN BACKWARD
OR NOT    P00148	// R_2nd DIE ALIGN FWD/BWD
AND LOAD
LOAD NOT  P00072	// R_2nd ALIGN CENTER FW
AND NOT   T1076	// R_2nd DIE ALIGN BACKWARD
OR LOAD
TON       T0580 400	// R_2nd DIE ALIGN FWD/BWD SN ALARM
; L401
LOAD      M00737	// R_2nd DIE ALIGN FWD/BWD SN ALARM
AND NOT   M00008	// LEFT RESET SW PLS
OR        T0580	// R_2nd DIE ALIGN FWD/BWD SN ALARM
OUT       M00737	// R_2nd DIE ALIGN FWD/BWD SN ALARM
; L403
LOAD      P00073	// R_2nd ALIGN LEFT FW
OR        P00149	// R_2nd DIE FPCB ALIGN FWD/BWD
LOAD      T1078	// R_2nd DIE FPCB ALIGN BACKWARD
OR NOT    P00149	// R_2nd DIE FPCB ALIGN FWD/BWD
AND LOAD
LOAD NOT  P00073	// R_2nd ALIGN LEFT FW
AND NOT   T1078	// R_2nd DIE FPCB ALIGN BACKWARD
OR LOAD
TON       T0581 400	// R_2nd DIE FPCB ALIGN FWD/BWD SN ALARM
; L406
LOAD      M00738	// R_2nd DIE FPCB ALIGN FWD/BWD SN ALARM
AND NOT   M00008	// LEFT RESET SW PLS
OR        T0581	// R_2nd DIE FPCB ALIGN FWD/BWD SN ALARM
OUT       M00738	// R_2nd DIE FPCB ALIGN FWD/BWD SN ALARM
; L408
LOAD      M0073E	// R_2nd DIE AUAc ¨úE©øN¨úi¢¯E
AND NOT   M00008	// LEFT RESET SW PLS
OR        M13110	// R_2nd DIE AUAc ¨úE©øN¨úi¢¯E
OUT       M0073E	// R_2nd DIE AUAc ¨úE©øN¨úi¢¯E

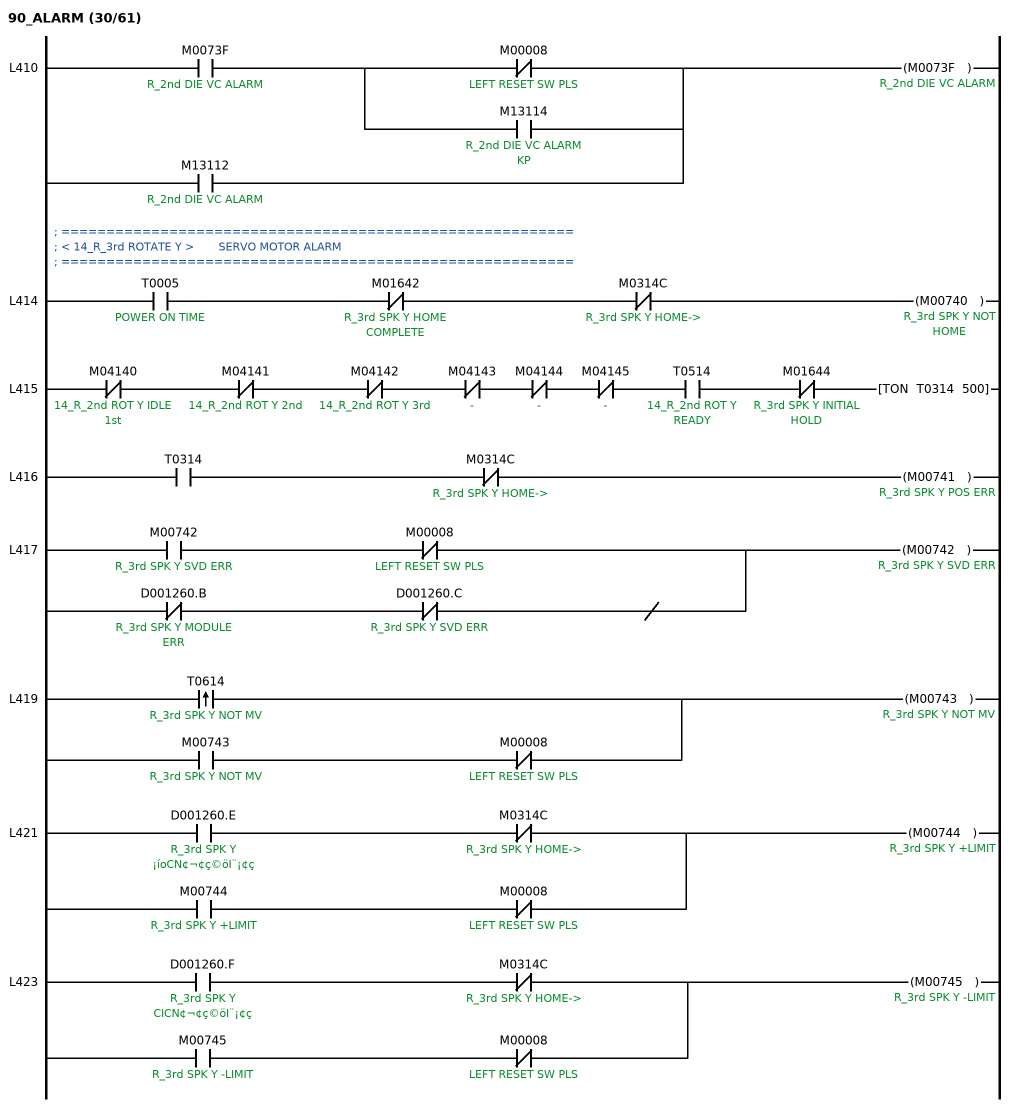
; L410
LOAD      M0073F	// R_2nd DIE VC ALARM
LOAD NOT  M00008	// LEFT RESET SW PLS
OR        M13114	// R_2nd DIE VC ALARM KP
AND LOAD
OR        M13112	// R_2nd DIE VC ALARM
OUT       M0073F	// R_2nd DIE VC ALARM
// =========================================================
// 
//        < 14_R_3rd ROTATE Y >       SERVO MOTOR ALARM
// 
// =========================================================
; L414
LOAD      T0005	// POWER ON TIME
AND NOT   M01642	// R_3rd SPK Y HOME COMPLETE
AND NOT   M0314C	// R_3rd SPK Y HOME->
OUT       M00740	// R_3rd SPK Y NOT HOME
; L415
LOAD NOT  M04140	// 14_R_2nd ROT Y IDLE 1st
AND NOT   M04141	// 14_R_2nd ROT Y 2nd
AND NOT   M04142	// 14_R_2nd ROT Y 3rd
AND NOT   M04143	// -
AND NOT   M04144	// -
AND NOT   M04145	// -
AND       T0514	// 14_R_2nd ROT Y READY
AND NOT   M01644	// R_3rd SPK Y INITIAL HOLD
TON       T0314 500
; L416
LOAD      T0314
AND NOT   M0314C	// R_3rd SPK Y HOME->
OUT       M00741	// R_3rd SPK Y POS ERR
; L417
LOAD      M00742	// R_3rd SPK Y SVD ERR
AND NOT   M00008	// LEFT RESET SW PLS
LOAD NOT  D001260.B	// R_3rd SPK Y MODULE ERR
AND NOT   D001260.C	// R_3rd SPK Y SVD ERR
NOT
OR LOAD
OUT       M00742	// R_3rd SPK Y SVD ERR
; L419
LOADP     T0614	// R_3rd SPK Y NOT MV
LOAD      M00743	// R_3rd SPK Y NOT MV
AND NOT   M00008	// LEFT RESET SW PLS
OR LOAD
OUT       M00743	// R_3rd SPK Y NOT MV
; L421
LOAD      D001260.E	// R_3rd SPK Y ¡íoCN¢¬¢ç©öI¨¡¢ç
AND NOT   M0314C	// R_3rd SPK Y HOME->
LOAD      M00744	// R_3rd SPK Y +LIMIT
AND NOT   M00008	// LEFT RESET SW PLS
OR LOAD
OUT       M00744	// R_3rd SPK Y +LIMIT
; L423
LOAD      D001260.F	// R_3rd SPK Y CICN¢¬¢ç©öI¨¡¢ç
AND NOT   M0314C	// R_3rd SPK Y HOME->
LOAD      M00745	// R_3rd SPK Y -LIMIT
AND NOT   M00008	// LEFT RESET SW PLS
OR LOAD
OUT       M00745	// R_3rd SPK Y -LIMIT

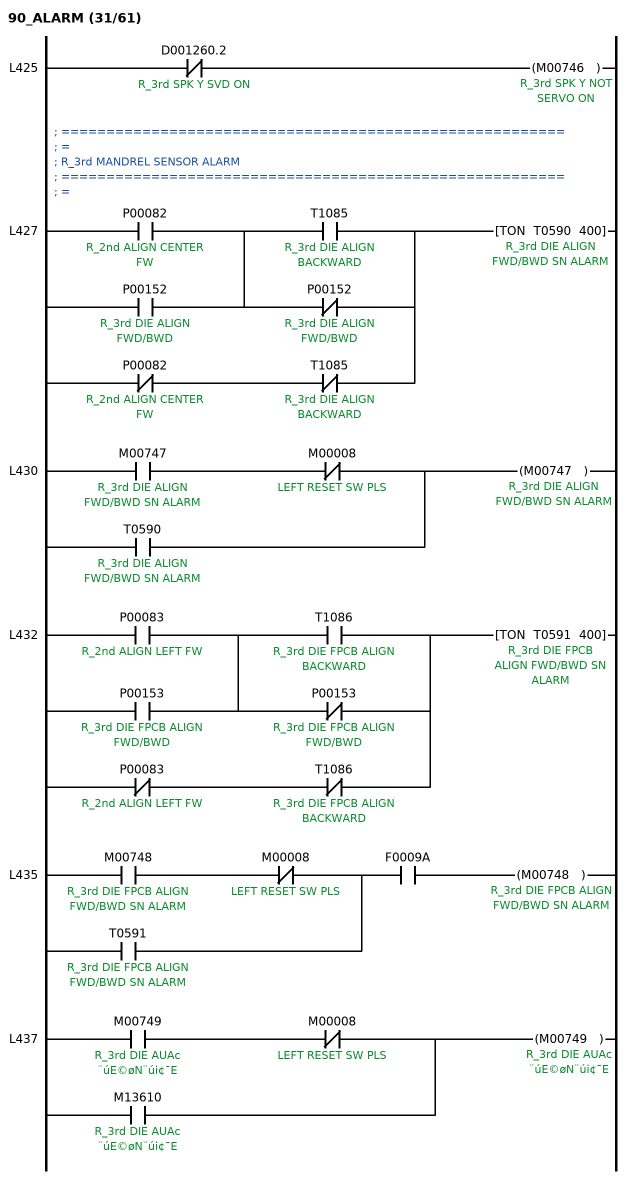
; L425
LOAD NOT  D001260.2	// R_3rd SPK Y SVD ON
OUT       M00746	// R_3rd SPK Y NOT SERVO ON
// =========================================================
// 
//        R_3rd MANDREL SENSOR ALARM
// 
// =========================================================
; L427
LOAD      P00082	// R_2nd ALIGN CENTER FW
OR        P00152	// R_3rd DIE ALIGN FWD/BWD
LOAD      T1085	// R_3rd DIE ALIGN BACKWARD
OR NOT    P00152	// R_3rd DIE ALIGN FWD/BWD
AND LOAD
LOAD NOT  P00082	// R_2nd ALIGN CENTER FW
AND NOT   T1085	// R_3rd DIE ALIGN BACKWARD
OR LOAD
TON       T0590 400	// R_3rd DIE ALIGN FWD/BWD SN ALARM
; L430
LOAD      M00747	// R_3rd DIE ALIGN FWD/BWD SN ALARM
AND NOT   M00008	// LEFT RESET SW PLS
OR        T0590	// R_3rd DIE ALIGN FWD/BWD SN ALARM
OUT       M00747	// R_3rd DIE ALIGN FWD/BWD SN ALARM
; L432
LOAD      P00083	// R_2nd ALIGN LEFT FW
OR        P00153	// R_3rd DIE FPCB ALIGN FWD/BWD
LOAD      T1086	// R_3rd DIE FPCB ALIGN BACKWARD
OR NOT    P00153	// R_3rd DIE FPCB ALIGN FWD/BWD
AND LOAD
LOAD NOT  P00083	// R_2nd ALIGN LEFT FW
AND NOT   T1086	// R_3rd DIE FPCB ALIGN BACKWARD
OR LOAD
TON       T0591 400	// R_3rd DIE FPCB ALIGN FWD/BWD SN ALARM
; L435
LOAD      M00748	// R_3rd DIE FPCB ALIGN FWD/BWD SN ALARM
AND NOT   M00008	// LEFT RESET SW PLS
OR        T0591	// R_3rd DIE FPCB ALIGN FWD/BWD SN ALARM
AND       F0009A
OUT       M00748	// R_3rd DIE FPCB ALIGN FWD/BWD SN ALARM
; L437
LOAD      M00749	// R_3rd DIE AUAc ¨úE©øN¨úi¢¯E
AND NOT   M00008	// LEFT RESET SW PLS
OR        M13610	// R_3rd DIE AUAc ¨úE©øN¨úi¢¯E
OUT       M00749	// R_3rd DIE AUAc ¨úE©øN¨úi¢¯E

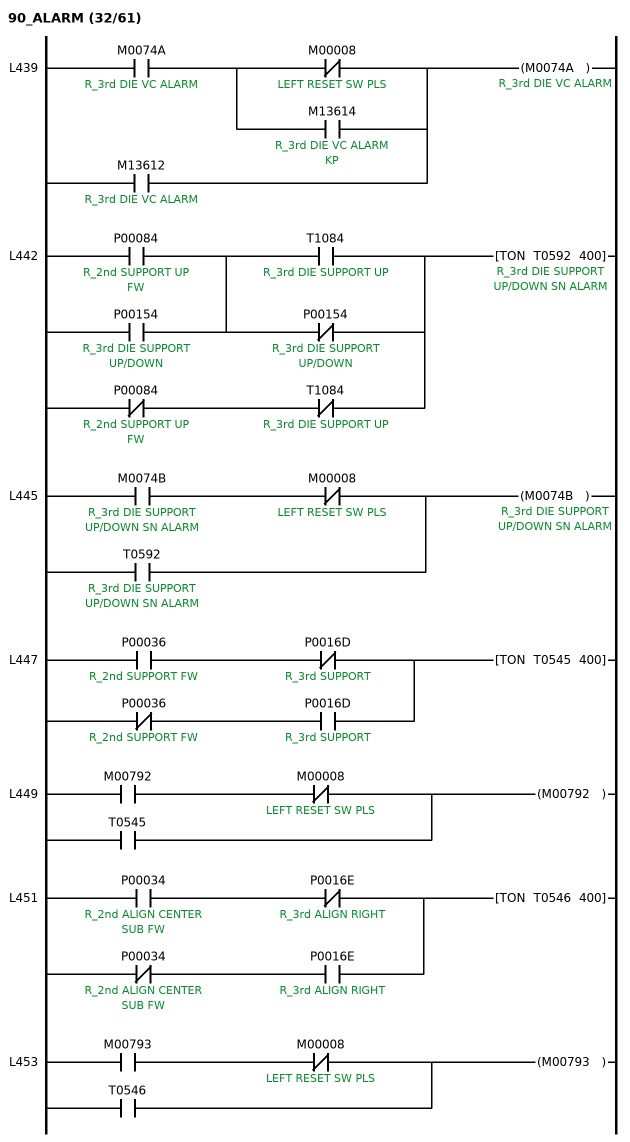
; L439
LOAD      M0074A	// R_3rd DIE VC ALARM
LOAD NOT  M00008	// LEFT RESET SW PLS
OR        M13614	// R_3rd DIE VC ALARM KP
AND LOAD
OR        M13612	// R_3rd DIE VC ALARM
OUT       M0074A	// R_3rd DIE VC ALARM
; L442
LOAD      P00084	// R_2nd SUPPORT UP FW
OR        P00154	// R_3rd DIE SUPPORT UP/DOWN
LOAD      T1084	// R_3rd DIE SUPPORT UP
OR NOT    P00154	// R_3rd DIE SUPPORT UP/DOWN
AND LOAD
LOAD NOT  P00084	// R_2nd SUPPORT UP FW
AND NOT   T1084	// R_3rd DIE SUPPORT UP
OR LOAD
TON       T0592 400	// R_3rd DIE SUPPORT UP/DOWN SN ALARM
; L445
LOAD      M0074B	// R_3rd DIE SUPPORT UP/DOWN SN ALARM
AND NOT   M00008	// LEFT RESET SW PLS
OR        T0592	// R_3rd DIE SUPPORT UP/DOWN SN ALARM
OUT       M0074B	// R_3rd DIE SUPPORT UP/DOWN SN ALARM
; L447
LOAD      P00036	// R_2nd SUPPORT FW
AND NOT   P0016D	// R_3rd SUPPORT
LOAD NOT  P00036	// R_2nd SUPPORT FW
AND       P0016D	// R_3rd SUPPORT
OR LOAD
TON       T0545 400
; L449
LOAD      M00792
AND NOT   M00008	// LEFT RESET SW PLS
OR        T0545
OUT       M00792
; L451
LOAD      P00034	// R_2nd ALIGN CENTER SUB FW
AND NOT   P0016E	// R_3rd ALIGN RIGHT
LOAD NOT  P00034	// R_2nd ALIGN CENTER SUB FW
AND       P0016E	// R_3rd ALIGN RIGHT
OR LOAD
TON       T0546 400
; L453
LOAD      M00793
AND NOT   M00008	// LEFT RESET SW PLS
OR        T0546
OUT       M00793

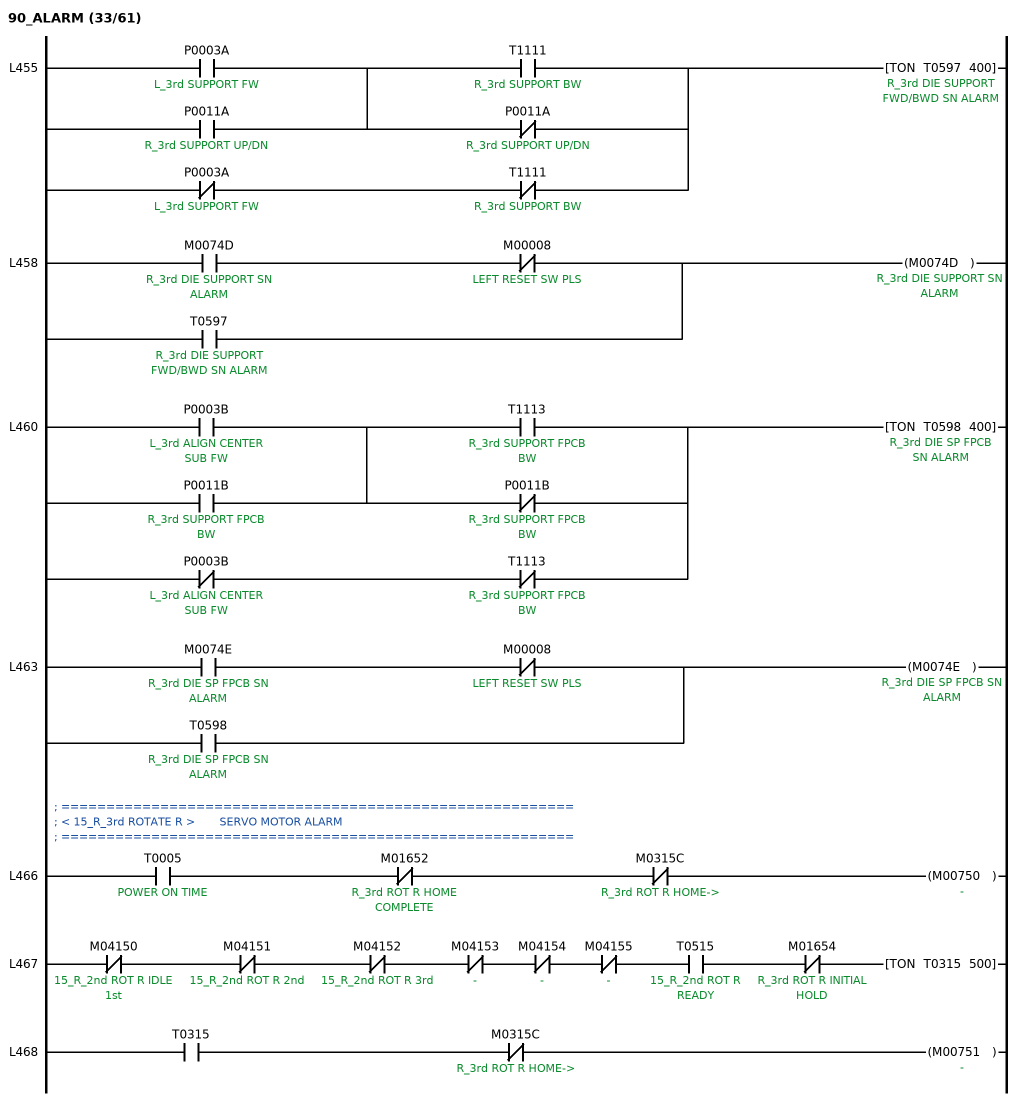
; L455
LOAD      P0003A	// L_3rd SUPPORT FW
OR        P0011A	// R_3rd SUPPORT UP/DN
LOAD      T1111	// R_3rd SUPPORT BW
OR NOT    P0011A	// R_3rd SUPPORT UP/DN
AND LOAD
LOAD NOT  P0003A	// L_3rd SUPPORT FW
AND NOT   T1111	// R_3rd SUPPORT BW
OR LOAD
TON       T0597 400	// R_3rd DIE SUPPORT FWD/BWD SN ALARM
; L458
LOAD      M0074D	// R_3rd DIE SUPPORT SN ALARM
AND NOT   M00008	// LEFT RESET SW PLS
OR        T0597	// R_3rd DIE SUPPORT FWD/BWD SN ALARM
OUT       M0074D	// R_3rd DIE SUPPORT SN ALARM
; L460
LOAD      P0003B	// L_3rd ALIGN CENTER SUB FW
OR        P0011B	// R_3rd SUPPORT FPCB BW
LOAD      T1113	// R_3rd SUPPORT FPCB BW
OR NOT    P0011B	// R_3rd SUPPORT FPCB BW
AND LOAD
LOAD NOT  P0003B	// L_3rd ALIGN CENTER SUB FW
AND NOT   T1113	// R_3rd SUPPORT FPCB BW
OR LOAD
TON       T0598 400	// R_3rd DIE SP FPCB SN ALARM
; L463
LOAD      M0074E	// R_3rd DIE SP FPCB SN ALARM
AND NOT   M00008	// LEFT RESET SW PLS
OR        T0598	// R_3rd DIE SP FPCB SN ALARM
OUT       M0074E	// R_3rd DIE SP FPCB SN ALARM
// =========================================================
// 
//        < 15_R_3rd ROTATE R >       SERVO MOTOR ALARM
// 
// =========================================================
; L466
LOAD      T0005	// POWER ON TIME
AND NOT   M01652	// R_3rd ROT R HOME COMPLETE
AND NOT   M0315C	// R_3rd ROT R HOME->
OUT       M00750	// -
; L467
LOAD NOT  M04150	// 15_R_2nd ROT R IDLE 1st
AND NOT   M04151	// 15_R_2nd ROT R 2nd
AND NOT   M04152	// 15_R_2nd ROT R 3rd
AND NOT   M04153	// -
AND NOT   M04154	// -
AND NOT   M04155	// -
AND       T0515	// 15_R_2nd ROT R READY
AND NOT   M01654	// R_3rd ROT R INITIAL HOLD
TON       T0315 500
; L468
LOAD      T0315
AND NOT   M0315C	// R_3rd ROT R HOME->
OUT       M00751	// -

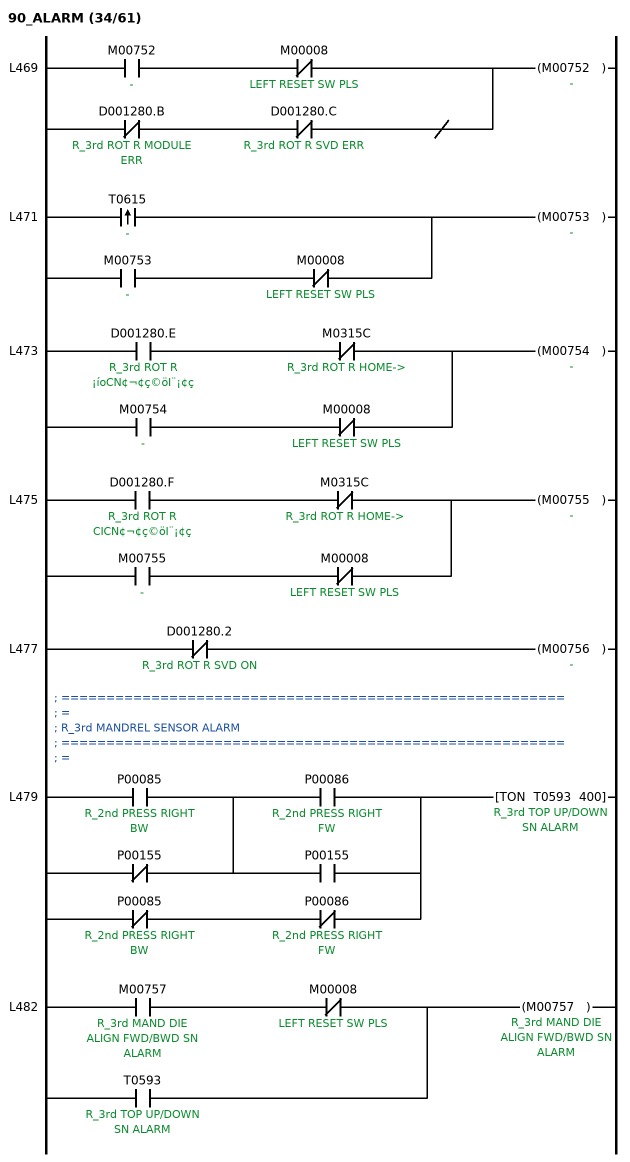
; L469
LOAD      M00752	// -
AND NOT   M00008	// LEFT RESET SW PLS
LOAD NOT  D001280.B	// R_3rd ROT R MODULE ERR
AND NOT   D001280.C	// R_3rd ROT R SVD ERR
NOT
OR LOAD
OUT       M00752	// -
; L471
LOADP     T0615	// -
LOAD      M00753	// -
AND NOT   M00008	// LEFT RESET SW PLS
OR LOAD
OUT       M00753	// -
; L473
LOAD      D001280.E	// R_3rd ROT R ¡íoCN¢¬¢ç©öI¨¡¢ç
AND NOT   M0315C	// R_3rd ROT R HOME->
LOAD      M00754	// -
AND NOT   M00008	// LEFT RESET SW PLS
OR LOAD
OUT       M00754	// -
; L475
LOAD      D001280.F	// R_3rd ROT R CICN¢¬¢ç©öI¨¡¢ç
AND NOT   M0315C	// R_3rd ROT R HOME->
LOAD      M00755	// -
AND NOT   M00008	// LEFT RESET SW PLS
OR LOAD
OUT       M00755	// -
; L477
LOAD NOT  D001280.2	// R_3rd ROT R SVD ON
OUT       M00756	// -
// =========================================================
// 
//        R_3rd MANDREL SENSOR ALARM
// 
// =========================================================
; L479
LOAD      P00085	// R_2nd PRESS RIGHT BW
OR NOT    P00155
LOAD      P00086	// R_2nd PRESS RIGHT FW
OR        P00155
AND LOAD
LOAD NOT  P00085	// R_2nd PRESS RIGHT BW
AND NOT   P00086	// R_2nd PRESS RIGHT FW
OR LOAD
TON       T0593 400	// R_3rd TOP UP/DOWN SN ALARM
; L482
LOAD      M00757	// R_3rd MAND DIE ALIGN FWD/BWD SN ALARM
AND NOT   M00008	// LEFT RESET SW PLS
OR        T0593	// R_3rd TOP UP/DOWN SN ALARM
OUT       M00757	// R_3rd MAND DIE ALIGN FWD/BWD SN ALARM

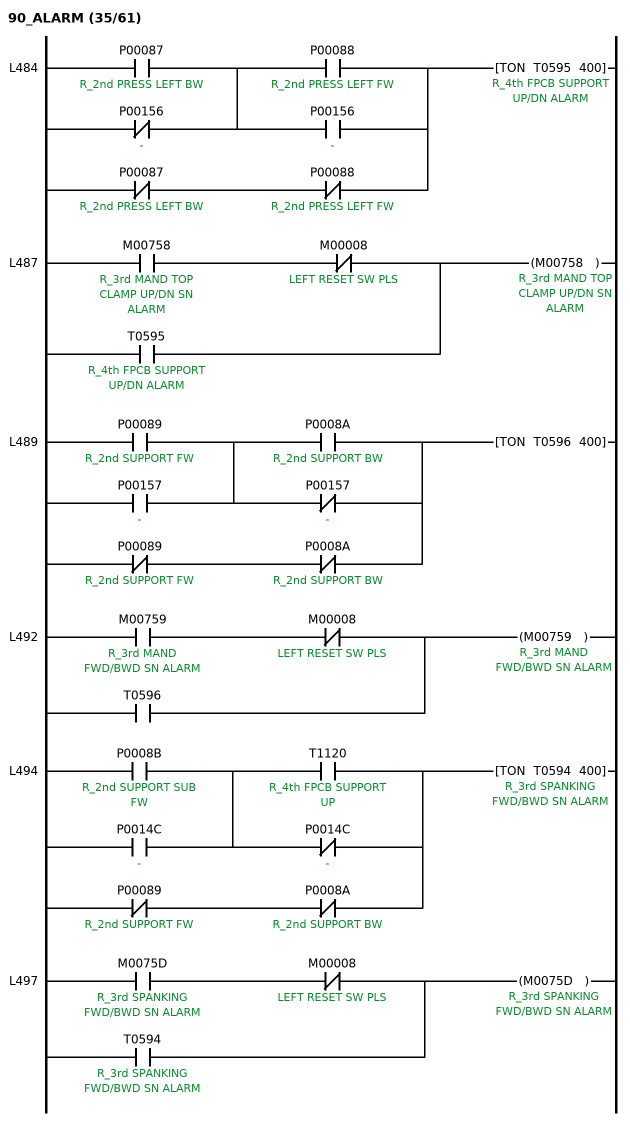
; L484
LOAD      P00087	// R_2nd PRESS LEFT BW
OR NOT    P00156	// -
LOAD      P00088	// R_2nd PRESS LEFT FW
OR        P00156	// -
AND LOAD
LOAD NOT  P00087	// R_2nd PRESS LEFT BW
AND NOT   P00088	// R_2nd PRESS LEFT FW
OR LOAD
TON       T0595 400	// R_4th FPCB SUPPORT UP/DN ALARM
; L487
LOAD      M00758	// R_3rd MAND TOP CLAMP UP/DN SN ALARM
AND NOT   M00008	// LEFT RESET SW PLS
OR        T0595	// R_4th FPCB SUPPORT UP/DN ALARM
OUT       M00758	// R_3rd MAND TOP CLAMP UP/DN SN ALARM
; L489
LOAD      P00089	// R_2nd SUPPORT FW
OR        P00157	// -
LOAD      P0008A	// R_2nd SUPPORT BW
OR NOT    P00157	// -
AND LOAD
LOAD NOT  P00089	// R_2nd SUPPORT FW
AND NOT   P0008A	// R_2nd SUPPORT BW
OR LOAD
TON       T0596 400
; L492
LOAD      M00759	// R_3rd MAND FWD/BWD SN ALARM
AND NOT   M00008	// LEFT RESET SW PLS
OR        T0596
OUT       M00759	// R_3rd MAND FWD/BWD SN ALARM
; L494
LOAD      P0008B	// R_2nd SUPPORT SUB FW
OR        P0014C	// -
LOAD      T1120	// R_4th FPCB SUPPORT UP
OR NOT    P0014C	// -
AND LOAD
LOAD NOT  P00089	// R_2nd SUPPORT FW
AND NOT   P0008A	// R_2nd SUPPORT BW
OR LOAD
TON       T0594 400	// R_3rd SPANKING FWD/BWD SN ALARM
; L497
LOAD      M0075D	// R_3rd SPANKING FWD/BWD SN ALARM
AND NOT   M00008	// LEFT RESET SW PLS
OR        T0594	// R_3rd SPANKING FWD/BWD SN ALARM
OUT       M0075D	// R_3rd SPANKING FWD/BWD SN ALARM

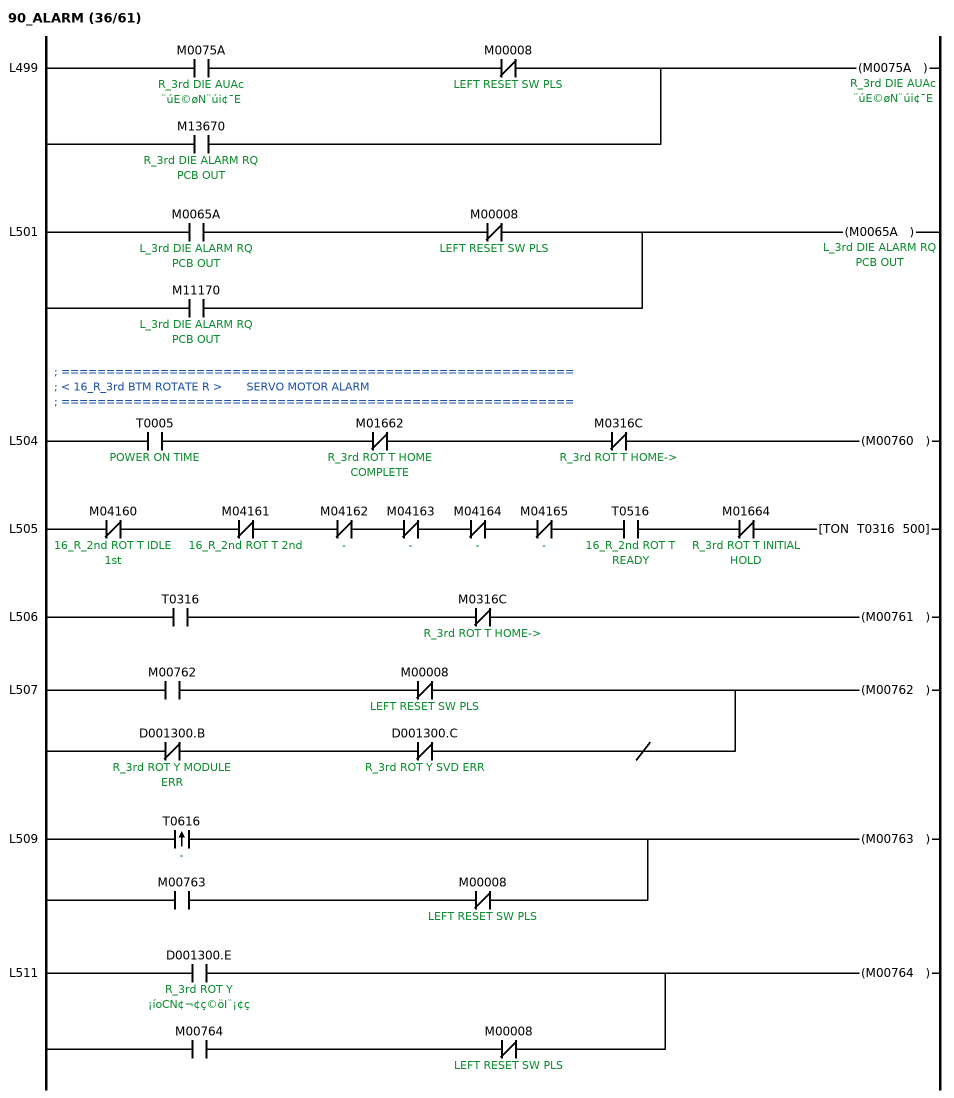
; L499
LOAD      M0075A	// R_3rd DIE AUAc ¨úE©øN¨úi¢¯E
AND NOT   M00008	// LEFT RESET SW PLS
OR        M13670	// R_3rd DIE ALARM RQ PCB OUT
OUT       M0075A	// R_3rd DIE AUAc ¨úE©øN¨úi¢¯E
; L501
LOAD      M0065A	// L_3rd DIE ALARM RQ PCB OUT
AND NOT   M00008	// LEFT RESET SW PLS
OR        M11170	// L_3rd DIE ALARM RQ PCB OUT
OUT       M0065A	// L_3rd DIE ALARM RQ PCB OUT
// =========================================================
// 
//        < 16_R_3rd BTM ROTATE R >       SERVO MOTOR ALARM
// 
// =========================================================
; L504
LOAD      T0005	// POWER ON TIME
AND NOT   M01662	// R_3rd ROT T HOME COMPLETE
AND NOT   M0316C	// R_3rd ROT T HOME->
OUT       M00760
; L505
LOAD NOT  M04160	// 16_R_2nd ROT T IDLE 1st
AND NOT   M04161	// 16_R_2nd ROT T 2nd
AND NOT   M04162	// -
AND NOT   M04163	// -
AND NOT   M04164	// -
AND NOT   M04165	// -
AND       T0516	// 16_R_2nd ROT T READY
AND NOT   M01664	// R_3rd ROT T INITIAL HOLD
TON       T0316 500
; L506
LOAD      T0316
AND NOT   M0316C	// R_3rd ROT T HOME->
OUT       M00761
; L507
LOAD      M00762
AND NOT   M00008	// LEFT RESET SW PLS
LOAD NOT  D001300.B	// R_3rd ROT Y MODULE ERR
AND NOT   D001300.C	// R_3rd ROT Y SVD ERR
NOT
OR LOAD
OUT       M00762
; L509
LOADP     T0616	// -
LOAD      M00763
AND NOT   M00008	// LEFT RESET SW PLS
OR LOAD
OUT       M00763
; L511
LOAD      D001300.E	// R_3rd ROT Y ¡íoCN¢¬¢ç©öI¨¡¢ç
LOAD      M00764
AND NOT   M00008	// LEFT RESET SW PLS
OR LOAD
OUT       M00764

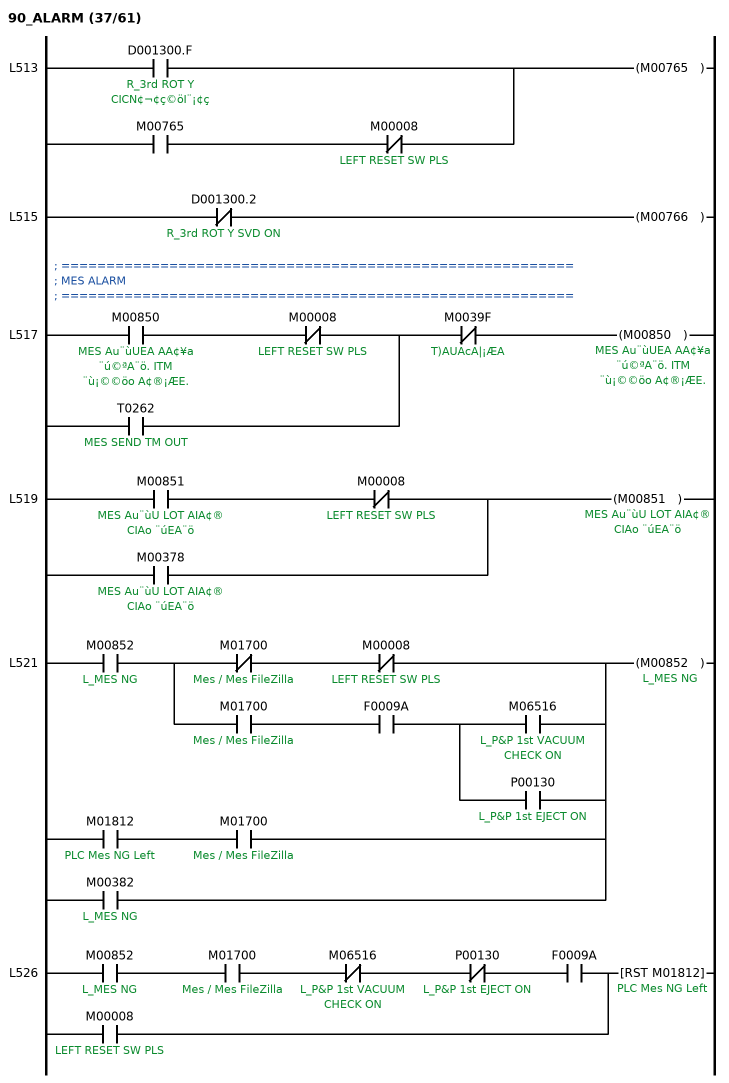
; L513
LOAD      D001300.F	// R_3rd ROT Y CICN¢¬¢ç©öI¨¡¢ç
LOAD      M00765
AND NOT   M00008	// LEFT RESET SW PLS
OR LOAD
OUT       M00765
; L515
LOAD NOT  D001300.2	// R_3rd ROT Y SVD ON
OUT       M00766
// =========================================================
// 
//        MES ALARM
// 
// =========================================================
; L517
LOAD      M00850	// MES Au¨ùUEA AA¢¥a ¨ú©ªA¨ö. ITM ¨ù¡©©öo A¢®¡ÆE.
AND NOT   M00008	// LEFT RESET SW PLS
OR        T0262	// MES SEND TM OUT
AND NOT   M0039F	// T)AUAcA|¡ÆA
OUT       M00850	// MES Au¨ùUEA AA¢¥a ¨ú©ªA¨ö. ITM ¨ù¡©©öo A¢®¡ÆE.
; L519
LOAD      M00851	// MES Au¨ùU LOT AIA¢® CIAo ¨úEA¨ö
AND NOT   M00008	// LEFT RESET SW PLS
OR        M00378	// MES Au¨ùU LOT AIA¢® CIAo ¨úEA¨ö
OUT       M00851	// MES Au¨ùU LOT AIA¢® CIAo ¨úEA¨ö
; L521
LOAD      M00852	// L_MES NG
LOAD NOT  M01700	// Mes / Mes FileZilla
AND NOT   M00008	// LEFT RESET SW PLS
LOAD      M01700	// Mes / Mes FileZilla
AND       F0009A
LOAD      M06516	// L_P&P 1st VACUUM CHECK ON
OR        P00130	// L_P&P 1st EJECT ON
AND LOAD
OR LOAD
AND LOAD
LOAD      M01812	// PLC Mes NG Left
AND       M01700	// Mes / Mes FileZilla
OR LOAD
OR        M00382	// L_MES NG
OUT       M00852	// L_MES NG
; L526
LOAD      M00852	// L_MES NG
AND       M01700	// Mes / Mes FileZilla
AND NOT   M06516	// L_P&P 1st VACUUM CHECK ON
AND NOT   P00130	// L_P&P 1st EJECT ON
AND       F0009A
OR        M00008	// LEFT RESET SW PLS
RST       M01812	// PLC Mes NG Left

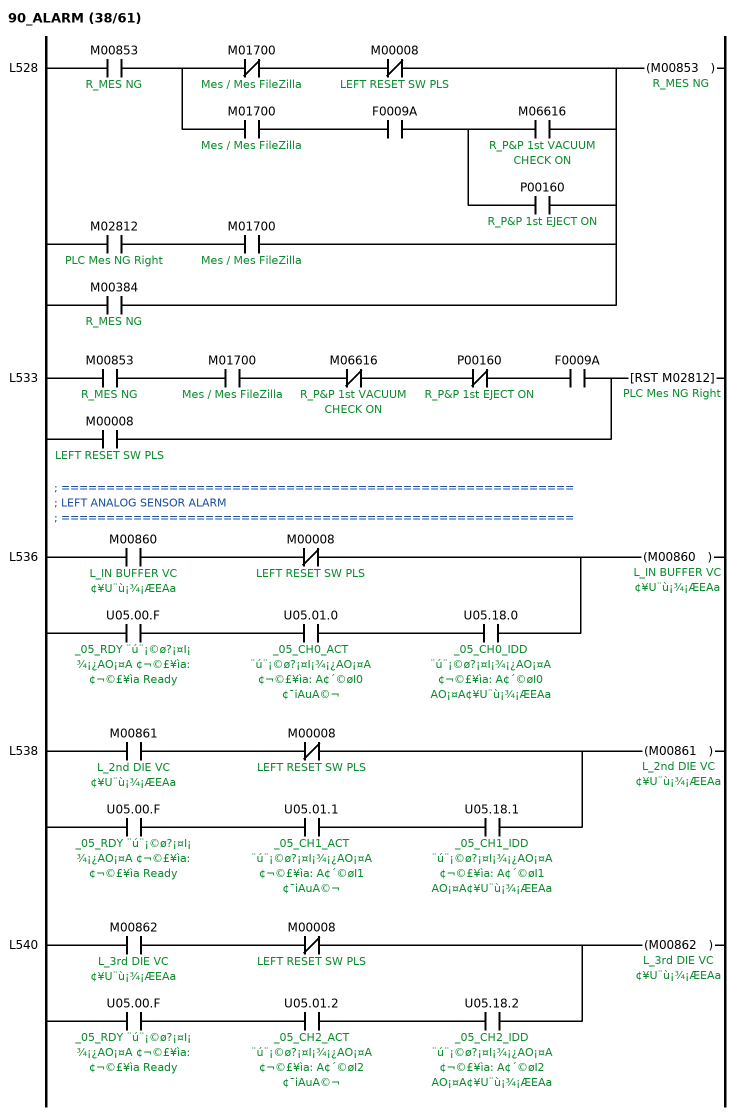
; L528
LOAD      M00853	// R_MES NG
LOAD NOT  M01700	// Mes / Mes FileZilla
AND NOT   M00008	// LEFT RESET SW PLS
LOAD      M01700	// Mes / Mes FileZilla
AND       F0009A
LOAD      M06616	// R_P&P 1st VACUUM CHECK ON
OR        P00160	// R_P&P 1st EJECT ON
AND LOAD
OR LOAD
AND LOAD
LOAD      M02812	// PLC Mes NG Right
AND       M01700	// Mes / Mes FileZilla
OR LOAD
OR        M00384	// R_MES NG
OUT       M00853	// R_MES NG
; L533
LOAD      M00853	// R_MES NG
AND       M01700	// Mes / Mes FileZilla
AND NOT   M06616	// R_P&P 1st VACUUM CHECK ON
AND NOT   P00160	// R_P&P 1st EJECT ON
AND       F0009A
OR        M00008	// LEFT RESET SW PLS
RST       M02812	// PLC Mes NG Right
// =========================================================
// 
//        LEFT ANALOG SENSOR ALARM
// 
// =========================================================
; L536
LOAD      M00860	// L_IN BUFFER VC ¢¥U¨ù¡¾¡ÆEAa
AND NOT   M00008	// LEFT RESET SW PLS
LOAD      U05.00.F	// _05_RDY ¨ú¨¡©ø?¡¤I¡¾¡¿AO¡¤A ¢¬©£¥ìa: ¢¬©£¥ìa Ready
AND       U05.01.0	// _05_CH0_ACT ¨ú¨¡©ø?¡¤I¡¾¡¿AO¡¤A ¢¬©£¥ìa: A¢´©øI0 ¢¯iAuA©¬
AND       U05.18.0	// _05_CH0_IDD ¨ú¨¡©ø?¡¤I¡¾¡¿AO¡¤A ¢¬©£¥ìa: A¢´©øI0 AO¡¤A¢¥U¨ù¡¾¡ÆEAa
OR LOAD
OUT       M00860	// L_IN BUFFER VC ¢¥U¨ù¡¾¡ÆEAa
; L538
LOAD      M00861	// L_2nd DIE VC ¢¥U¨ù¡¾¡ÆEAa
AND NOT   M00008	// LEFT RESET SW PLS
LOAD      U05.00.F	// _05_RDY ¨ú¨¡©ø?¡¤I¡¾¡¿AO¡¤A ¢¬©£¥ìa: ¢¬©£¥ìa Ready
AND       U05.01.1	// _05_CH1_ACT ¨ú¨¡©ø?¡¤I¡¾¡¿AO¡¤A ¢¬©£¥ìa: A¢´©øI1 ¢¯iAuA©¬
AND       U05.18.1	// _05_CH1_IDD ¨ú¨¡©ø?¡¤I¡¾¡¿AO¡¤A ¢¬©£¥ìa: A¢´©øI1 AO¡¤A¢¥U¨ù¡¾¡ÆEAa
OR LOAD
OUT       M00861	// L_2nd DIE VC ¢¥U¨ù¡¾¡ÆEAa
; L540
LOAD      M00862	// L_3rd DIE VC ¢¥U¨ù¡¾¡ÆEAa
AND NOT   M00008	// LEFT RESET SW PLS
LOAD      U05.00.F	// _05_RDY ¨ú¨¡©ø?¡¤I¡¾¡¿AO¡¤A ¢¬©£¥ìa: ¢¬©£¥ìa Ready
AND       U05.01.2	// _05_CH2_ACT ¨ú¨¡©ø?¡¤I¡¾¡¿AO¡¤A ¢¬©£¥ìa: A¢´©øI2 ¢¯iAuA©¬
AND       U05.18.2	// _05_CH2_IDD ¨ú¨¡©ø?¡¤I¡¾¡¿AO¡¤A ¢¬©£¥ìa: A¢´©øI2 AO¡¤A¢¥U¨ù¡¾¡ÆEAa
OR LOAD
OUT       M00862	// L_3rd DIE VC ¢¥U¨ù¡¾¡ÆEAa

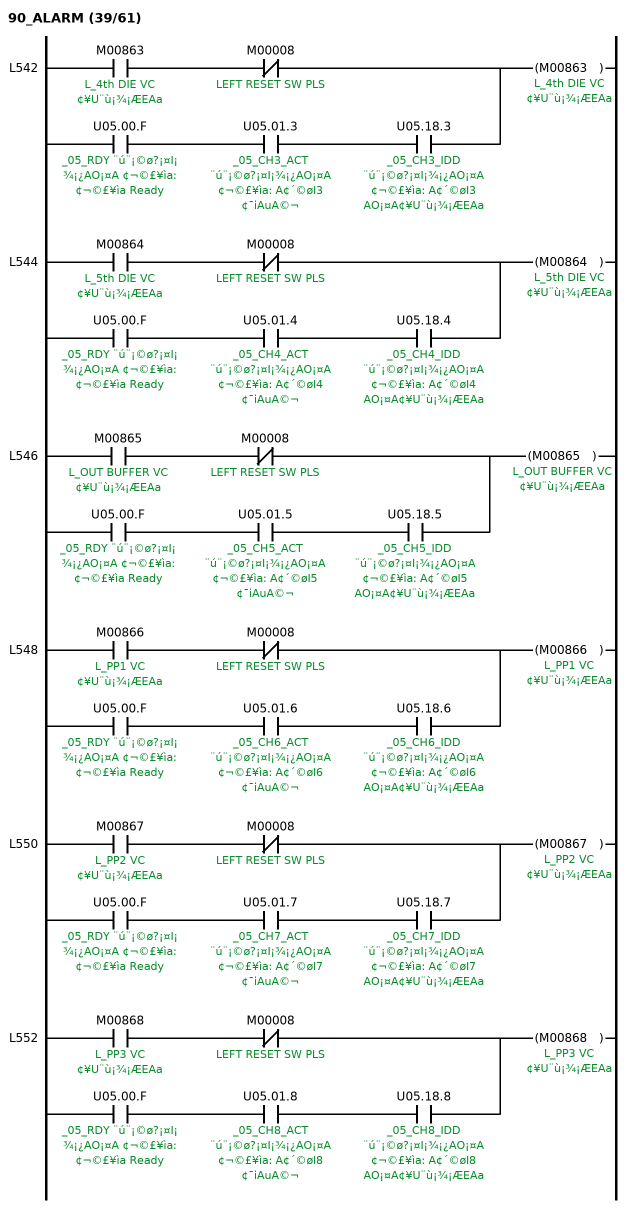
; L542
LOAD      M00863	// L_4th DIE VC ¢¥U¨ù¡¾¡ÆEAa
AND NOT   M00008	// LEFT RESET SW PLS
LOAD      U05.00.F	// _05_RDY ¨ú¨¡©ø?¡¤I¡¾¡¿AO¡¤A ¢¬©£¥ìa: ¢¬©£¥ìa Ready
AND       U05.01.3	// _05_CH3_ACT ¨ú¨¡©ø?¡¤I¡¾¡¿AO¡¤A ¢¬©£¥ìa: A¢´©øI3 ¢¯iAuA©¬
AND       U05.18.3	// _05_CH3_IDD ¨ú¨¡©ø?¡¤I¡¾¡¿AO¡¤A ¢¬©£¥ìa: A¢´©øI3 AO¡¤A¢¥U¨ù¡¾¡ÆEAa
OR LOAD
OUT       M00863	// L_4th DIE VC ¢¥U¨ù¡¾¡ÆEAa
; L544
LOAD      M00864	// L_5th DIE VC ¢¥U¨ù¡¾¡ÆEAa
AND NOT   M00008	// LEFT RESET SW PLS
LOAD      U05.00.F	// _05_RDY ¨ú¨¡©ø?¡¤I¡¾¡¿AO¡¤A ¢¬©£¥ìa: ¢¬©£¥ìa Ready
AND       U05.01.4	// _05_CH4_ACT ¨ú¨¡©ø?¡¤I¡¾¡¿AO¡¤A ¢¬©£¥ìa: A¢´©øI4 ¢¯iAuA©¬
AND       U05.18.4	// _05_CH4_IDD ¨ú¨¡©ø?¡¤I¡¾¡¿AO¡¤A ¢¬©£¥ìa: A¢´©øI4 AO¡¤A¢¥U¨ù¡¾¡ÆEAa
OR LOAD
OUT       M00864	// L_5th DIE VC ¢¥U¨ù¡¾¡ÆEAa
; L546
LOAD      M00865	// L_OUT BUFFER VC ¢¥U¨ù¡¾¡ÆEAa
AND NOT   M00008	// LEFT RESET SW PLS
LOAD      U05.00.F	// _05_RDY ¨ú¨¡©ø?¡¤I¡¾¡¿AO¡¤A ¢¬©£¥ìa: ¢¬©£¥ìa Ready
AND       U05.01.5	// _05_CH5_ACT ¨ú¨¡©ø?¡¤I¡¾¡¿AO¡¤A ¢¬©£¥ìa: A¢´©øI5 ¢¯iAuA©¬
AND       U05.18.5	// _05_CH5_IDD ¨ú¨¡©ø?¡¤I¡¾¡¿AO¡¤A ¢¬©£¥ìa: A¢´©øI5 AO¡¤A¢¥U¨ù¡¾¡ÆEAa
OR LOAD
OUT       M00865	// L_OUT BUFFER VC ¢¥U¨ù¡¾¡ÆEAa
; L548
LOAD      M00866	// L_PP1 VC ¢¥U¨ù¡¾¡ÆEAa
AND NOT   M00008	// LEFT RESET SW PLS
LOAD      U05.00.F	// _05_RDY ¨ú¨¡©ø?¡¤I¡¾¡¿AO¡¤A ¢¬©£¥ìa: ¢¬©£¥ìa Ready
AND       U05.01.6	// _05_CH6_ACT ¨ú¨¡©ø?¡¤I¡¾¡¿AO¡¤A ¢¬©£¥ìa: A¢´©øI6 ¢¯iAuA©¬
AND       U05.18.6	// _05_CH6_IDD ¨ú¨¡©ø?¡¤I¡¾¡¿AO¡¤A ¢¬©£¥ìa: A¢´©øI6 AO¡¤A¢¥U¨ù¡¾¡ÆEAa
OR LOAD
OUT       M00866	// L_PP1 VC ¢¥U¨ù¡¾¡ÆEAa
; L550
LOAD      M00867	// L_PP2 VC ¢¥U¨ù¡¾¡ÆEAa
AND NOT   M00008	// LEFT RESET SW PLS
LOAD      U05.00.F	// _05_RDY ¨ú¨¡©ø?¡¤I¡¾¡¿AO¡¤A ¢¬©£¥ìa: ¢¬©£¥ìa Ready
AND       U05.01.7	// _05_CH7_ACT ¨ú¨¡©ø?¡¤I¡¾¡¿AO¡¤A ¢¬©£¥ìa: A¢´©øI7 ¢¯iAuA©¬
AND       U05.18.7	// _05_CH7_IDD ¨ú¨¡©ø?¡¤I¡¾¡¿AO¡¤A ¢¬©£¥ìa: A¢´©øI7 AO¡¤A¢¥U¨ù¡¾¡ÆEAa
OR LOAD
OUT       M00867	// L_PP2 VC ¢¥U¨ù¡¾¡ÆEAa
; L552
LOAD      M00868	// L_PP3 VC ¢¥U¨ù¡¾¡ÆEAa
AND NOT   M00008	// LEFT RESET SW PLS
LOAD      U05.00.F	// _05_RDY ¨ú¨¡©ø?¡¤I¡¾¡¿AO¡¤A ¢¬©£¥ìa: ¢¬©£¥ìa Ready
AND       U05.01.8	// _05_CH8_ACT ¨ú¨¡©ø?¡¤I¡¾¡¿AO¡¤A ¢¬©£¥ìa: A¢´©øI8 ¢¯iAuA©¬
AND       U05.18.8	// _05_CH8_IDD ¨ú¨¡©ø?¡¤I¡¾¡¿AO¡¤A ¢¬©£¥ìa: A¢´©øI8 AO¡¤A¢¥U¨ù¡¾¡ÆEAa
OR LOAD
OUT       M00868	// L_PP3 VC ¢¥U¨ù¡¾¡ÆEAa

